# B&R Automation Studio project TD52 (part 86)

#### DirAirInj.var - Local variables
```iecst
(********************************************************************
 * COPYRIGHT -- INNIO Company
 ********************************************************************
 * Program: DirectAirInjection
 * File: DirectAirInjection.var
 * Author: 212754567
 * Created: May 15, 2019
 ********************************************************************
 * Local variables of program DirectAirInjection
 ********************************************************************)

VAR
	xDTGetTime : DTGetTime;
	iDAI_Sec_Act : UDINT; (* direct air injection actual operation time [s] *)
	DT_DAI_Start : DATE_AND_TIME; (* direct air injection starting date and time *)
	xTON_DAI_V_Open_Fault : TON; (* direct air injection inlet valve opening fault delay*)
	xTON_DAI_V_Close_Fault : TON; (* direct air injection inlet valve closing fault delay*)
	xSR_DAI_V_Close_Fault : SR; (* set/reset close fault for direct air injection inlet valve *)
	xSR_DAI_V_Open_Fault : SR; (* set/reset open fault for direct air injection inlet valve *)
	xTOF_DAI_V_Dem : TOF; (* shutdown delay for shut off valve *)
	xTOF_Pr_AirStarter_Tank_Lo : TOF; (* delay enable signal from start tank pressure *)
END_VAR

VAR CONSTANT

END_VAR
```

### Program Logical/EngineController/misf_ctr_EC (IEC) - + misfire monitoring and power reduction

- misf_ctr.st (not readable text: treated as protected, skipped)

#### misf_ctr.var
```iecst
VAR
	bMisfElectrical : BOOL; (* memory for electrical misfire *)
	slMisfIntern : DINT; (* internal integrator for el. misf. *)
	TP_MisfBlink : TP; (* blink pulse for visu. misfiring *)
	ssMisfInt : INT;
	TON_Misfire_Relase : TON;
END_VAR
```

### Program Logical/EngineController/misf_det_EC (IEC) - + detection of misfire using actual power

- misf_det.st (not readable text: treated as protected, skipped)

#### misf_det.var
```iecst
VAR
	ssPowerAuss1 : INT; (* last actual power in permill nom. *)
	FILTER_ActPower : FILTER; (* FUB filter actual power T=30 msec. *)
	bNewAuss : BOOL; (* TRUE= new misfire can be detected *)
	slHilf1 : DINT; (* max.zul.Steilheit von P_ist KW/sec *)
END_VAR
```

### Program Logical/EngineController/MsgEC (IEC) - + Engine Controller Messages

- MsgECCyclic.st (not readable text: treated as protected, skipped)

- MsgECInit.st (not readable text: treated as protected, skipped)

#### MsgEC.var
```iecst
VAR
	iAdrMM2AmmBase : UDINT;
	iAdrAmmBase2MM : UDINT;
	xMsg1080 : Msg;
	xMsg3217 : Msg;
	xMsg1044 : Msg;
	xMsg1049 : Msg;
	xMsg1153 : Msg;
	xMsg3542 : Msg;
	xMsg2061 : Msg;
	xMsg2062 : Msg;
	xMsg2063 : Msg;
	xMsg2064 : Msg;
	xMsg2065 : Msg;
	xMsg2066 : Msg;
	xMsg2067 : Msg;
	xMsg2068 : Msg;
	xMsg2069 : Msg;
	xMsg2070 : Msg;
	xMsg2071 : Msg;
	xMsg2072 : Msg;
	xMsg2073 : Msg;
	xMsg2074 : Msg;
	xMsg2075 : Msg;
	xMsg2076 : Msg;
	xMsg2077 : Msg;
	xMsg2078 : Msg;
	xMsg2079 : Msg;
	xMsg2080 : Msg;
	xMsg2339 : Msg;
	xMsg2365 : Msg;
	xMsg3408 : Msg;
	xMsg3409 : Msg;
	xTON_FG_MSATM : TON;
	FG_MSATM : BOOL;
	xMsg1047 : Msg;
	xMsg3212 : Msg;
	xMsg3099 : Msg;
	xMsg2084 : Msg;
	xMsg1192 : Msg;
	xMsg2514 : Msg;
	xMsg2515 : Msg;
	xMsg2516 : Msg;
	xMsg2517 : Msg;
	xMsg2522 : Msg;
	xMsg2523 : Msg;
	xMsg3348 : Msg;
	xMsg3583 : Msg;
	xMsg3584 : Msg;
	xMsg3529 : Msg;
	xMsg3585 : Msg;
	xMsg3564 : Msg;
	xMsg3371 : Msg;
	xMsg3372 : Msg;
	xMsg3373 : Msg;
	xMsg3374 : Msg;
	bRPSA7_624 : BOOL;
	xTOF_1080_rel : TOF;
	xMsg3586 : Msg;
	FG_ABMW : BOOL; (*Freigabe Abweichung Mittelwert*)
	ton_ABMW : TON;
	xMsg2294 : Msg;
	xMsg2283 : Msg;
	xMsg9216 : Msg;
	xMsg2287 : Msg;
	xMsg2290 : Msg;
	xMsg2262 : Msg;
	xMsg2282 : Msg;
	xMsg2274 : Msg;
	xMsg2588 : Msg;
	xMsg2577 : Msg;
	xMsg2583 : Msg;
	b2880 : BOOL;
	b2881 : BOOL;
	i : USINT;
	iNum_b2880 : USINT;
	iNum_b2881 : USINT;
	xMsg3382 : Msg;
	xMsg2518 : Msg;
	xMsg2519 : Msg;
	xMsg2520 : Msg;
	xMsg2521 : Msg;
	xMsg2562 : Msg;
	xMsg3555 : Msg;
	xMsg3556 : Msg;
	xMsg3557 : Msg;
	xMsg3558 : Msg;
	xMsg2470 : Msg;
	xMsg2471 : Msg;
	xMsg2487 : Msg; (*warning for recommend leanox adjustment*)
	xMsg2488 : Msg; (*warning for mandatory leanox adjustment*)
	xMsg9246 : Msg;
	xMsg2328 : Msg;
	xMsg2329 : Msg;
	xMsg9247 : Msg;
	xMsg9248 : Msg;
	xMsg9253 : Msg; (*warning for Leanox 2 saturation *)
	xMsg9288 : Msg; (* warning: measuring signal failure, temperature direct air injection *)
	xMsg9289 : Msg; (* warning: measuring signal failure, pressure before direct air injection shut off valve  *)
	xMsg9290 : Msg; (* warning: measuring signal failure, pressure before direct air injection control valve bank A *)
	xMsg9291 : Msg; (* warning: measuring signal failure, pressure before direct air injection control valve bank B *)
	xMsg9292 : Msg; (* warning: direct air injection shut off valve failure at closing*)
	xMsg9293 : Msg; (* warning: direct air injection shut off valve failure at opening*)
	xMsg9294 : Msg; (* warning: direct air injection circuit breaker tripped  *)
	xMsg9295 : Msg; (* warning: direct air injection tank pressure low*)
	xMsg9296 : Msg; (* warning: direct air injection control valve bank A failure *)
	xMsg9297 : Msg; (* warning: direct air injection control valve bank B failure *)
	xMsg9298 : Msg; (* warning: direct air injection pressure before shut off valve high *)
	xMsg9299 : Msg; (* warning: direct air injection failure *)
	xMsg9039 : Msg; (* warning: direct air injection active*)
	xMsg9040 : Msg; (* warning: direct air injection inactive*)
	xMsg9312 : Msg; (* Generator frequency too low in mains parallel operation *)
	xMsg9313 : Msg; (* Generator frequency too high in mains parallel operation *)
	xMsg9329 : Msg; (* p2 sensor signal for GEN2 controller missing *)
	xMsg2975 : Msg; (* Fast-Gas-Quality-Change-Function is running *)
	xMsg9047 : Msg; (* operating message: target load reached *)
	xMsg9349 : Msg; (* Grid Code FRT functionality contains wrong parameter *)
	xMsg9053 : Msg; (* operating message: SCR inlet temperature controller active *)
	xMsg9054 : Msg; (* operating message: SCR inlet temperature controller inactive *)
	xMsg9055 : Msg; (* operating message: th. reactor start time reduction - operating cycle started *)
	xMsg9056 : Msg; (* operating message: th. reactor start time reduction - operating cycle completed *)
	xMsg9065 : Msg; (* operating message: Isolated operation - Grid status detection *)
	xMsg9095 : Msg; (* operating message: GEN2 lambda offset stopped *)
	xMsg2765 : Msg; (* warning: PI optimizer opening duration offset in limitation *)
	xMsg3268 : Msg; (* operating message: PI optimizer opening duration offset in limitation *)
	xMsg9373 : Msg; (* warning: PI-Optimization not allowed *)
	xMsg9078 : Msg; (* operating message: PI-Optimization not allowed *)
	xMsg2768 : Msg; (* gas humidity measuring signal failure *)
	xMsg2880 : Msg;	(** B2880: Cylinder exhaust gas temperature positive deviation from average value *)
	xMsg2881 : Msg;	(** B2881: Cylinder exhaust gas temperature negative deviation from average value *)
	xMsg2970 : Msg;	(** B2970: Exhaust gas temperature inclination maximum at cylinder head *)
	xMsg1293 : Msg;	(** B1293: Engine map automatically loaded *)
	xMsg2814 : Msg;	(** B2814: Open durance Port Injection high *)
	xMsg2874 : Msg;	(** B2874: Safety layer sensor failure *)
	xMsg2802 : Msg;	(** B2802: Cylinder pressure sensor measuring signal failure *)
	xMsg2808 : Msg;	(** B2808: Maximum positive deviation of average cylinder peak pressure *)
	xMsg2825 : Msg;	(** B2825: Cylinder peak pressure high Warning *)
	xMsg2826 : Msg;	(** B2826: Cylinder peak pressure high *)
	xMsg2849 : Msg;	(** B2849: Misfiring failure *)
	xMsg2145 : Msg;	(** B2145: Ignition point reduction PBC *)
	xMsg2876 : Msg;	(** B2876: Misfire controller shutdown *)
	xMsg2882 : Msg;	(** B2882: Balancer map deleted *)
	xMsg2883 : Msg;	(** B2883: Balancer map saved *)
	xMsg2960 : Msg;	(** B2960: Ignition point reduction by Cylinder Peak Pressure Integrator *)
	xMsg2141 : Msg;	(** B2141: ignition point optimization *)
	xMsg3238 : Msg;	(** B3238: Positive deviation of cylinder x from average high *)
	xMsg3239 : Msg;	(** B3239: Negative deviation of cylinder x from average high *)
	xMsg3247 : Msg;	(** B3247: TECJET step of gas volume high *)
	xMsg3248 : Msg;	(** B3248: TECJET fuel gas volume high *)
	xMsg3285 : Msg;	(** B3285: exh. gas temp. measuring signal failure *)
	xMsg3295 : Msg;	(** B3295: operation message max. exhaust temperature *)
	xMsg2831 : Msg;	(** B2831: Low Voltage Ride Through Event  --> bBM_GrC_Event *)
	xMsg2832 : Msg;	(** B2832: Mains failure + Generator Pole slip -->  bBM_PoleSlip *)
	xMsg2833 : Msg;	(** B2833: Mains failure + dynamic rotor angle maximum --> bBM_disconnect_dynAng*)
	xMsg2834 : Msg;	(** B2834: Mains failure + static rotor angle maximum -->  bBM_disconnect_staticAng*)
	xMsg2835 : Msg;	(** B2835: Mains failure + leading power factor operation -->bBM_disconnect_CapMode*)
	xMsg2836 : Msg;	(** B2836: Mains failure maintenance request, reserve *)
	xMsg2837 : Msg;	(** B2837: Mains failure + dynamic rotor angle minimum --> bBM_disconnect_dynAng_Min*)
	xMsg2838 : Msg;	(** B2838: Mains failure + electric power to low --> bBM_disconnect_Power*)
	xMsg2839 : Msg;	(** B2839: Mains failure + U(t)< *)
	xMsg9068 : Msg;	(** B9068: Fault ride trougth event  --> bBM_FRT_Event *)
	xMsg9071 : Msg;	(** B9071: Low Voltage Ride Through Event simulated --> bBM_GrC_Event_Sim *)
	xMsg2840 : Msg;	(** B2840: Spare *)
	xMsg2841 : Msg;	(** B2841: Emergency shutdown on gas valves *)
	xMsg2846 : Msg;	(** B2846: Fast power reduction due to auto-ignition *)
	xMsg2852 : Msg;	(** B2852: Turbocharger surge *)
	xMsg2165 : Msg;	(** B2165: Power limitation by air humidity - low limit *)(* Humidity Package *)
	xMsg2166 : Msg;	(** B2166: Air humidity charge temperature offset active *)(* Humidity Package *)
	xMsg2894 : Msg;	(** B2894: Engine map is missing *)
	xMsg1294 : Msg;	(** B1294: performing WG check *)
	xMsg1299 : Msg;	(** B1299: optimizer map changed *)
	xMsg2187 : Msg;	(** B2187: Commissioning mode on *)
	xMsg2188 : Msg;	(** B2188: Commissioning mode off *)
	xMsg2897 : Msg;	(** B2897: Boost pressure out of range*)
	xMsg2929 : Msg;	(** B2929: Cylinder IMEP deviation from average value *)
	xMsg2930 : Msg;	(** B2930: PI optimization required *)
	xMsg2937 : Msg;	(* B2937 LEANOX new adjusted *)
	xMsg2938 : Msg;	(* B2938 Combustion chamber cleaning performed *)
	xMsg2986 : Msg;	(* B2986 Leanox 2 Active - operator message *)
	xMsg2987 : Msg;	(* B2987 Leanox 2 Not Active - operator message *)
	xMsg9388 : Msg; (* warning: combustion anomaly detected *)
	xMsg9392 : Msg; (*warning: CAN wastegate bank A Actuator Failure *)
	xMsg9393 : Msg; (*warning: CAN wastegate bank B Actuator Failure *)
	xMsg9394 : Msg; (*warning: CAN wastegate bank A System Warnings *)
	xMsg9395 : Msg; (*warning: CAN wastegate bank B System Warnings *)
	xMsg2380 : Msg; (*alarm: CAN wastegate bank A CAN Communication Error *)
	xMsg2381 : Msg; (*alarm: CAN wastegate bank B CAN Communication Error *)
END_VAR
```

### Program Logical/EngineController/OUT_EC_TC1 (IEC) - + Engine Controller output task TC1

- OUT_EC_TC1.st (not readable text: treated as protected, skipped)

### Program Logical/EngineController/OUT_EngCtr (IEC) - + Engine Controller output task

- OUT_EngCtr.st (not readable text: treated as protected, skipped)

### Program Logical/EngineController/exhaust_EC (IEC) - + monitoring the exhaust gas temperatures

- exhaustCyclic.st (not readable text: treated as protected, skipped)

- exhaustInit.st (not readable text: treated as protected, skipped)

#### exhaust.var
```iecst
VAR
	FilterCylTemp : ARRAY[0..24] OF FILTER;
	CylTemp_1 : ARRAY[0..24] OF INT;
	ssDeltaCylTemp : INT;
	ABMWN_acttime : ARRAY[0..24] OF UINT; (* 1 hour timer neg. avg. dev. *)
	ABMWN_time : ARRAY[0..24] OF tABMW_time; (* error time memory neg. avg. dev. *)
	ABMWP_acttime : ARRAY[0..24] OF UINT; (* 1 nhour timer pos. avg. dev. *)
	ABMWP_time : ARRAY[0..24] OF tABMW_time; (* error time memory pos. avg. dev. *)
	AmmSeqABMWN : AmmSequence; (* FUB AmmSeq. neg. dev. avg. *)
	AmmSeqABMWP : AmmSequence; (* FUB AmmSeq. pos. dev. avg *)
	AmmSeqATMA : AmmSequence;
	AmmSeqMSAGT : AmmSequence;
	slTempAverage : DINT; (* sum up for average temp. *)
	ssTempLimitNeg : INT; (* cyl.temp. limit negative *)
	ssTempLimitPos : INT; (* cyl.temp. limit positive *)
	ssTempZylMax : INT; (* cyl.temp. maximum value *)
	ssTempZylMin : INT; (* cyl.temp. minimum value *)
	t_zylMax : INT; (* maximal temp. accord. to AN_GW40 *)
	TON_ABMWN : TON; (*reset timer for neg. avg. dev.*)
	TON_ABMWP : TON; (*reset timer for pos. avg. dev.*)
	TON_CheckTemp : TON; (* delay of exh.temp. monitoring *)
	TON_Cycle : TON; (* cycle time for program duration *)
	ucABMWNCount : USINT; (* nbr. of cyl. with neg. deviation *)
	ucABMWPCount : USINT; (* nr. of cyl. with pos. deviation *)
	ucAnzahlZylABWMN : USINT; (* number of cyl. with divagance neg. *)
	ucAverageCount : USINT; (* average # of cylinder counter *)
	ucCylinderCount : USINT; (* cylinder number counter for loops *)
	ucTimeCount : USINT; (* loop counter time memory *)
	usABMWNtime : UINT; (* 1 hour timer neg. avg. dev. *)
	usABMWPtime : UINT; (* 1 hour timer pos. avg. dev. *)
	usTempMaxCount : ARRAY[0..24] OF USINT; (* counter delay max. cyl. temp. *)
	usTempNegCount : ARRAY[0..24] OF USINT; (* counter delay of neg. deviation *)
	usTempPosCount : ARRAY[0..24] OF USINT; (* counter delay of pos. deviation *)
	xHys_EGT_Avg : GR_MAXR;
	xRamp_PRed_EGT_Avg : RAMPE_R;
	t_zyl_mw : INT;
	TOF_HiContSkip : ARRAY[0..25] OF TOF;
	xSimPID_EGT : SimPID4 := (0);
	LCRScal_EG_Max : LCRScal;
	FILTER_EG_Max : FILTER_R;
	TP_ExhLim_FS : TP;
	TON_TempMax_Ext : ARRAY[0..24] OF TON;
	xTON_TempMax_Ext_TrStRed : ARRAY[0..24] OF TON;
	bEngine_Stopped : BOOL;
	TP_bZylAusfall : TP;
	t_zyl_old : ARRAY[0..24] OF INT;
	bEG_Grad : ARRAY[0..24] OF BOOL;
	rT_dTExhMon_ITPComp : REAL; (*TExh compensation at later ITP values (positive values for increasing temp. at retarding) [K/Â°CA]*)
	bdTExhMonTrip : ARRAY[0..24] OF BOOL; (*TRUE = TExhMon trip detected for cylinder*)
	rTsample : REAL; (*task sample time*)
	rdTExh_Misfire : REAL := 20; (*delta temperature from reference to misfire limit [°C]*)
	AmmSeqdTExhMon : AmmSequence;
	bPCGVmonInit : BOOL;
	iCnt_PCGV_class1_Mem : ARRAY[0..24] OF UINT;
	iCnt_PCGV_class2_Mem : ARRAY[0..24] OF UINT;
	iCnt_PCGV_class3_Mem : ARRAY[0..24] OF UINT;
	iCnt_PCGV_class4_Mem : ARRAY[0..24] OF UINT;
	xGR_MINR_t_zyl : ARRAY[0..24] OF GR_MINR;
	xR_TRIG_EGT_PRed : R_TRIG;
	bMSAGT_Warn : ARRAY[0..24] OF BOOL; (*Set the exhaust gas temperature sensor warning*)
	xFILTER_EG_Cyl : ARRAY[0..24] OF FILTER_R;
	iFilt_EG_Cyl : UINT := 5;
	rFILTER_EG_Cyl_old : ARRAY[0..24] OF REAL;
	xGR_MAXR_t_zyl_BackfPrev : ARRAY[0..24] OF GR_MAXR;
	rT_EG_Grad_Hyst : REAL := 0;
	xTP_Ena_BackfPrev : TP;
	rPos_CBV_Release_BackfPrev : REAL := 0.05;
	xMEDIAN_EG_Filt : RMEDIAN24 := (0);
	rGrad_EG_Median : REAL;
	rGrad_EG_Median_old : REAL;
	xTON_t_zyl_BackfPrev : ARRAY[0..24] OF TON;
	tiBackPrevOnDelay : TIME := T#3s;
	rGrad_EG_Filt : ARRAY[0..24] OF REAL;
	rGrad_EG_Filt_Diff2Median : ARRAY[0..24] OF REAL;
	rGrad_EG_Median_Vect : ARRAY[0..24] OF REAL;
	xF_TRIG_bHoldBackfPrev : F_TRIG;
	bBlockBackfPrev : BOOL;
	rP_Act_Norm_BackfPrevOFF : REAL := 0.8;
	bW9388_Array1 : ARRAY[0..24] OF BOOL;
	bW9388_Array2 : ARRAY[0..24] OF BOOL;
	bW9388_Array_Compare : ARRAY[0..24] OF BOOL;
	AmmSeqCombAnomaly : AmmSequence;
	xR_TRIG_bW9388_Array : R_TRIG;
	ucEventCounter : USINT; (*Event counter for loops *)
	xTOF_ZylAusfall : ARRAY[0..20] OF TOF := [21((0))]; (*Timer für Events Zylinderausfall*)
	bTrigZylAusfall : BOOL := 0;
	iZylAusfallErrCout : INT := 0;
	bZylAusfall_test : BOOL := 0;
	rTi_EGT_NegDev : REAL := 180.0; (*Exhaust temperature negative deviation max. duration*)
	rTi_EGT_NegDev_TimeDur : REAL := 180.0; (*Exhauxt temperature negaitve deviation monitoring time duration*)
	iCnt_EGT_NegDev_max : INT := 10; (*Exhaust temperature negative deviation max. count*)
END_VAR
```

### Program Logical/EngineController/dyn_GR (IEC) - + GridCode

- Dyn_GRCyclic.st (not readable text: treated as protected, skipped)

- Dyn_GRInit.st (not readable text: treated as protected, skipped)

#### Dyn_GR.var - Local variables
```iecst
(********************************************************************
 * COPYRIGHT -- INNIO Company
 ********************************************************************
 * Program: dyn_GR
 * File:
 * Author:
 * Created:
 ********************************************************************
 * Local variables of program
 ********************************************************************)
VAR
	bSimulate : BOOL; (*simulation variable*) (* OldName: bSimulate; Cycle:2; *)
	xF_TRIG_IgnOFF : F_TRIG; (* 0 *) (* OldName: F_TRIG_IgnOFF; Cycle:2; *)
	xF_TRIG_VoltRecovPlusT : F_TRIG; (* 0 *) (* OldName: F_TRIG_VoltRecovPlusT; Cycle:2; *)
	xF_TRIG_GCEventPeriode_PA : F_TRIG; (* 0 *) (* OldName: F_TRIG_GCEventPeriode_PA; Cycle:2; *)
	xF_TRIG_GCEvent : F_TRIG; (* 0 *) (* OldName: F_TRIG_GCEvent; Cycle:2; *)
	rN_GrC_Speed : REAL; (* speed for Grid Code calculations *) (* OldName: ssGridCodeSpeed; Cycle:2; *)
	rI_GrC_Lim : REAL; (* Grid Code current limit in [A ]*) (* OldName: ssCurrentLimit; Cycle:2; *)
	rPhase_Ang_Const : REAL; (* constant for phase angel calculation *) (* OldName: fPhaseAngleConst; Cycle:2; *)
	rN_GrC_SpeedChange_Lim : REAL; (* speed change limit for Grid Code event detection *) (* OldName: ssGridCodeSpeedChangeLimit; Cycle:2; *)
	r_Eng_Cyc : REAL; (* Length of motor cycle [ms]*) (* OldName: ssMotorzyklus; Cycle:2; *)
	rU_GrC_Lim : REAL; (* Grid Code voltage limit in [V ]*) (* OldName: ssVoltageLimit; Cycle:2; *)
	rN_Ign_Int : REAL; (* speed ignition [1/min] *) (* OldName: n_Ign_INTERNAL; Cycle:2; *)
	xR_TRIG_IgnOFFON : R_TRIG; (* 0 *) (* OldName: R_TRIG_IgnOFFON; Cycle:2; *)
	xR_TRIG_IgnOFF : R_TRIG; (* 0 *) (* OldName: R_TRIG_IgnOFF; Cycle:2; *)
	xR_TRIG_Wait : R_TRIG; (* 0 *) (* OldName: R_TRIG_Wart; Cycle:2; *)
	xR_TRIG_GCE_Power : R_TRIG; (* 0 *) (* OldName: R_TRIG_GCE_Power; Cycle:2; *)
	xR_TRIG_GCE : R_TRIG; (* 0 *) (* OldName: R_TRIG_GCE; Cycle:2; *)
	xR_TRIG_GCEvent : R_TRIG; (* 0 *) (* OldName: R_TRIG_GCEvent; Cycle:2; *)
	tLam_Ada : TIME; (* 0 *) (* OldName: tLambdaAdabt; Cycle:2; *)
	tLeanoxCtrMan : TIME; (* 0 *) (* OldName: tLeanoxCtrMan; Cycle:2; *)
	tEventPulse : TIME; (* Pulse time for Grid Code event *) (* OldName: tEventPulse; Cycle:2; *)
	tHilfsbetriebeTripOFF : TIME; (* 0 *) (* OldName: tHilfsbetriebeTripOFF; Cycle:2; *)
	tPumpErk : TIME; (* Dauer fuer Aktivierung der Pumperkennung *) (* OldName: tPumpErk; Cycle:2; *)
	tTimeAfterVoltRecov : TIME; (* Zeit nach der, nach Wiederkehr der Spannung, die Zuendung eingeschaltet wird *) (* OldName: tTimeAfterVoltRecov; Cycle:2; *)
	tLeanoxErrorOFF : TIME; (* tLeanoxErrorOFF : TIME; *) (* OldName: tLeanoxErrorOFF; Cycle:2; *)
	tPowerFIX : TIME; (* Dauer Leistungsfixierung bei GCEvent / time Power setting *) (* OldName: tPowerFIX; Cycle:2; *)
	xTOF_GCEventPeriode_PA : TOF; (* *) (* OldName: TOF_GCEventPeriode_PA; Cycle:2; *)
	xTOF_GrC_EventPeriode : TOF; (* No phase angle reset for 1 sec. in case of Grid Code event *) (* OldName: TOF_GirdCodeEventPeriode; Cycle:2; *)
	xTOF_Netp : TOF; (* wait 5 sec. after disconnection from grid to disable the simulation flag *) (* OldName: TOF_Netp; Cycle:2; *)
	xTON_Netp : TON; (* wait 5 sec, after switch to netprallel before use average speed *) (* OldName: xTON_Netp; Cycle:2; *)
	xTON_PoleSlip : TON; (* 0 *) (* OldName: xTON_PoleSlip; Cycle:2; *)
	xTON_ConstGenPF : TON; (* TON check const generator power factor *) (* OldName: TON_ConstGenPF; Cycle:2; *)
	xTON_AvgPeriode : TON; (* time period for average calculation *) (* OldName: TON_AvgPeriode; Cycle:2; *)
	xTON_ConstGenCurr : TON; (*TON check const generator current *) (* OldName: TON_ConstGenCurr; Cycle:2; *)
	xTON_ConstGenFreq : TON; (* 0 *) (* OldName: TON_ConstGenFreq; Cycle:2; *)
	xTP_GrC_Event : TP; (* 0 *) (* OldName: TP_GridCodeEvent; Cycle:2; *)
	xTP_GrC_Event_BM : TP; (* 0 *) (* OldName: TP_GridCodeEvent_BM; Cycle:2; *)
	xTP_GrC_Event_Sim_BM : TP; (* 0 *)
	xTP_GCE_PumpErk : TP; (* 0 *) (* OldName: TP_GCE_PumpErk; Cycle:2; *)
	xTP_GCE_LeanoxErr : TP; (* 0 *) (* OldName: TP_GCE_LeanoxErr; Cycle:2; *)
	xTP_GCE_PowerFIX : TP; (* 0 *) (* OldName: TP_GCE_PowerFIX; Cycle:2; *)
	xTP_VoltRecov : TP; (* 0 *) (* OldName: TP_VoltRecov; Cycle:2; *)
	xTP_Wart : TP; (* 0 *) (* OldName: TP_Wart; Cycle:2; *)
	xTP_PoleSlip : TP; (* 0 *) (* OldName: TP_PoleSlip; Cycle:2; *)
	xTP_IgnOffPump : TP; (* 0 *) (* OldName: TP_IgnOffPump; Cycle:2; *)
	xTP_IgnOnVoltRecov : TP; (* 0 *) (* OldName: TP_IgnOnVoltRecov ; Cycle:2; *)
	xTP_GCE_LeanoxCtr : TP; (* 0 *) (* OldName: TP_GCE_LeanoxCtr; Cycle:2; *)
	xTP_Disc_dynAng_Min_BM : TP; (* 0 *) (* OldName: TP_disconnect_dynAngle_Min_BM; Cycle:2; *)
	xTP_Disc_Power_BM : TP; (* 0 *) (* OldName: TP_disconnect_Power_BM; Cycle:2; *)
	xTP_Disc_dynAng_BM : TP; (* 0 *) (* OldName: TP_disconnect_dynAngle_BM; Cycle:2; *)
	xTP_GCE_Power : TP; (* 0 *) (* OldName: TP_GCE_Power; Cycle:2; *)
	xTP_Disc_CapMode_BM : TP; (* 0 *) (* OldName: TP_disconnect_CapMode_BM; Cycle:2; *)
	xTP_GCE_HBTrip : TP; (* 0 *) (* OldName: TP_GCE_HBTrip; Cycle:2; *)
	xTP_GCE_Lam_Ada : TP; (* 0 *) (* OldName: TP_GCE_LambdaAdabt; Cycle:2; *)
	xTP_GCE : TP; (* 0 *) (* OldName: TP_GCE; Cycle:2; *)
	xTP_DO_GRIDCODE_DCON_TC1 : TP; (* 0 *) (* OldName: TP_DO_GRIDCODE_DCON_TC1; Cycle:2; *)
	xTP_Disc_staticAng_BM : TP; (* 0 *) (* OldName: TP_disconnect_staticAngle_BM; Cycle:2; *)
	xTP_GCE_FIXAct : TP; (* 0 *) (* OldName: TP_GCE_FIXAct; Cycle:2; *)
	xTP_CurrentChange : TP; (* 0 *) (* OldName: TP_CurrentChange; Cycle:2; *)
	xTP_SpeedChange : TP; (* 0 *) (* OldName: TP_SpeedChange; Cycle:2; *)
	xTP_VoltageLow : TP; (* 0 *) (* OldName: TP_VoltageLow; Cycle:2; *)
	b_GrC_VoltageLow : BOOL; (* TRUE if Grid Code event low voltage is detected *) (* OldName: TP_VoltRecov; Cycle:2; *)
	bRel_PA_RESET : BOOL; (* TRUE = PA after 350ms reset *) (* OldName: bFREIGABE_PA_RESET; Cycle:2; *)
	bGrC_Disc_Cap : BOOL; (* Decoupling when capacitance operating in Grid Code Event *) (* OldName: bGC_disconnect_Cap; Cycle:2; *)
	bGrC_Disc_DynAng : BOOL; (* Decouple when static + dynamic angle during GCEvents> Limit*) (* OldName: bGC_disconnect_DynAngle; Cycle:2; *)
	bGrC_Disc_DynAng_Min : BOOL; (* Decouple when static + dynamic angle during GCEvents <Limit*(-1) and voltage below Limi *) (* OldName: bGC_disconnect_DynAngle_Min; Cycle:2; *)
	bGrC_Disc_Power : BOOL; (* Decouple when power < Limit when entering the GC events *) (* OldName: bGC_disconnect_Power; Cycle:2; *)
	bGrC_Disc_StaticAng : BOOL; (* Decouple when static angle already when entering the GC Events> Limit *) (* OldName: bGC_disconnect_StaticAngle; Cycle:2; *)
	bGrC_DO_int : BOOL; (* 0 *) (* OldName: bGC_DO_int; Cycle:2; *)
	bGrC_LamAdabt : BOOL; (* TRUE = Lambda-Adaption aktiv (BR<6) bei BR6 sowieso aktiv LVIC Gasmengenberechnung *) (* OldName: bGC_LambdaAdabt; Cycle:2; *)
	bGrC_LeanoxCtrMAN : BOOL; (* TRUE = Leanox Regler ist im Handbetrieb (GCEvent) *) (* OldName: bGC_LeanoxCtrMAN; Cycle:2; *)
	bGrC_LeanoxCtrMan : BOOL; (* TRUE = Leanox Regler bei GCEvent fuer def. Zeit in Hand *) (* OldName: bGC_LeanoxCtrMan; Cycle:2; *)
	bGrC_LeanoxErrOFF : BOOL; (* TRUE = LoxAbw. A1080 wird bei GCEvent blockiert *) (* OldName: bGC_LeanoxErrOFF; Cycle:2; *)
	bGrC_PowerFIX_Akt : BOOL; (* TRUE = Leistungsfixierung bei GridCodeEvent im eng_ctr aktiv *) (* OldName: bGC_PowerFIX_Akt; Cycle:2; *)
	bGrC_CurrentChange : BOOL; (* TRUE if generator current change is above limit *) (* OldName: bGridCodeCurrentChange; Cycle:2; *)
	bGrC_CurrentChange_Mer : BOOL; (*cuurent chagne merker*) (* OldName: bGridCodeCurrentChange_MERKER; Cycle:2; *)
	bGrC_SpeedChange : BOOL; (* TRUE if Grid Code event speed change is detected *) (* OldName: bGridCodeSpeedChange; Cycle:2; *)
	bGrC_SpeedChange_Mer : BOOL; (*speed change merker*) (* OldName: bGridCodeSpeedChange_MERKER; Cycle:2; *)
	bGrC_Missf : BOOL; (* Switch off the ignition active /TRUE = Zuendungausschalten AKTIV *) (* OldName: bGridMissf; Cycle:2; *)
	bIgnOFF_Mer : BOOL; (* Merker fuer Zuendung AUS *) (* OldName: bIgnOFF_MERKER; Cycle:2; *)
	bIgnON_Mer : BOOL; (* Merker fuer Zuendung EIN *) (* OldName: bIgnON_MERKER; Cycle:2; *)
	bCap : BOOL; (* TRUE = capacitive Engine Run *) (* OldName: bKap; Cycle:2; *)
	bNFilter2 : BOOL; (* TRUE = Avg 2 Perioden | FALSE = 3 Perioden *) (* OldName: bNFilter2; Cycle:2; *)
	bPoleSlip : BOOL; (* TRUE if pole slip detected *) (* OldName: bPoleSlip; Cycle:2; *)
	bPoleSlip_INT : BOOL; (*Pole slip detection*) (* OldName: bPoleSlip_INT; Cycle:2; *)
	bTP_GrC_Event : BOOL; (* TP TRUE Grid Code event *) (* OldName: bTP_GridCodeEvent; Cycle:2; *)
	r_CosPhi : REAL; (* generator cos phi *) (* OldName: fCosPhi; Cycle:2; *)
	r_Phi : REAL; (* generator phi in radian *) (* OldName: fPhi; Cycle:2; *)
	r_Divisor : REAL; (* divisor for polar wheel angle calculation *) (* OldName: fDivisor; Cycle:2; *)
	xFILTER_cosphi : FILTER_R; (*Filter fuer Cos Phi - da Messung im Falle eines Events nicht plausibel*) (* OldName: FILTER_cosphi; Cycle:2; *)
	r_PhaseAng_OFF : REAL; (* dyn. Winkel bei dem die Zuendung AUSgeschalten wird [°] *) (* OldName: fPhaseAngelIgnOFF; Cycle:2; *)
	r_PhaseAng_ON : REAL; (* dyn. Winkel bei dem die Zuendung wieder EINgeschalten wird [°] *) (* OldName: fPhaseAngelIgnON; Cycle:2; *)
	r_PolarWheelAng : REAL; (* calcualted polar wheel angle in degree *) (* OldName: fPolarWheelAngle; Cycle:2; *)
	r_PolarWheelAng_GC : REAL; (* 0 *) (* OldName: fPolarWheelAngle_GC; Cycle:2; *)
	r_Xqo : REAL; (* 0 *) (* OldName: fXqo; Cycle:2; *)
	i_IgnOFF_Time : INT; (* Ignition off aktiv, counter wie lange *) (* OldName: IgnOFF_Time; Cycle:2; *)
	i_IgnOFF_TimeMin : INT; (* 0 *) (* OldName: IgnOFF_TimeMIN; Cycle:2; *)
	iMissfCyl_old_GC : UDINT; (* 0 *) (* OldName: MissfCyl_old_GC; Cycle:2; *)
	rN_Ign1_Avg : REAL; (* avarage speed ignition [1/min] *) (* OldName: n_Ign1_Avg; Cycle:2; *)
	rN_Ign1_old : REAL; (* old speed ignition [1/min] *) (* OldName: n_Ign1_old; Cycle:2; *)
	rN_Ign1_old2 : REAL; (* old speed ignition [1/min] *) (* OldName: n_Ign1_old2; Cycle:2; *)
	rN_GrC_SpeedSumm : REAL; (* speed average sample summ *) (* OldName: slGridCodeSpeedSumm; Cycle:2; *)
	rN_AvgSpeed : REAL; (* 100 sample speed average used for phase angle calcualtion *) (* OldName: ssAvgSpeed; Cycle:2; *)
	rN_AvgSpeed1 : REAL; (* ast sample speed average used for phase angle calcualtion *) (* OldName: ssAvgSpeed1; Cycle:2; *)
	rN_AvgSpeed2 : REAL; (* last sample speed average used for phase angle calcualtion *) (* OldName: ssAvgSpeed2; Cycle:2; *)
	rCnT_GrC_CurrentChange_PULSE : REAL; (* current change puls counter *) (* OldName: ssGCCurrentChange_PULSE_COUNTER; Cycle:2; *)
	rI_GrC_CurrentChange_PULSE_Lim : REAL; (* 0 *) (* OldName: ssGCCurrentChange_PULSE_LIMIT; Cycle:2; *)
	rCnt_GrC_SpeedChange_PULSE : REAL; (* 0 *) (* OldName: ssGCSpeedChange_PULSE_COUNTER; Cycle:2; *)
	rN_GrC_SpeedChange_PULSE_Lim : REAL; (* 0 *) (* OldName: ssGCSpeedChange_PULSE_LIMIT; Cycle:2; *)
	rIgn_Cnt_Off : REAL; (* ignition OFF activate / Zuendung AUS aktiv -> zaehlen wie lange *) (* OldName: ssIgnAUS_Countms; Cycle:2; *)
	rCnt_IGN_Off : REAL; (*Counter for ignition OFF / Counter fuer Zuendung AUS *) (* OldName: ssIGNOFF_COUNTER; Cycle:2; *)
	rCnt_IGN_On : REAL; (*Counter for ignition ON / Counter fuer Zuendung EIN *) (* OldName: ssIGNON_COUNTER; Cycle:2; *)
	r_IL1_Change : REAL; (* change of generator current L1 since last task cycle *) (* OldName: ssIL1Change; Cycle:2; *)
	r_IL2_Change : REAL; (* change of generator current L2 since last task cycle *) (* OldName: ssIL2Change; Cycle:2; *)
	r_IL3_Change : REAL; (* change of generator current L3 since last task cycle *) (* OldName: ssIL3Change; Cycle:2; *)
	r_IL1_Last : REAL; (* Generator current phase 1 from last cycle *) (* OldName: ssLastIL1; Cycle:2; *)
	r_IL2_Last : REAL; (* Generator current phase 2 from last cycle *) (* OldName: ssLastIL2; Cycle:2; *)
	r_IL3_Last : REAL; (* Generator current phase 3 from last cycle *) (* OldName: ssLastIL3; Cycle:2; *)
	r_CosPhi_Last : REAL; (* last power factor *) (* OldName: ssLastCosPhi; Cycle:2; *)
	r_GrC_LastSpeed : REAL; (*speed from last cycle *) (* OldName: ssLastGridCodeSpeed; Cycle:2; *)
	r_Freq_Last : REAL; (*last generator frequency *) (* OldName: usLastFreq; Cycle:2; *)
	iSpeedOption : USINT; (*speed options*) (* OldName: ucSpeedOption; Cycle:2; *)
	bGrC_PumpErk : BOOL; (* TRUE = Pumperkennung bei GC Events aktiv *) (* OldName: bGC_PumpErk; Cycle:2; *)
	iMMUSynchFWVers : ARRAY[0..2] OF UINT; (* Firmware version MMUsynch *) (* OldName: usMMUSynchFWVers; Cycle:2; *)
	iFreqConv : UINT; (* Conversion fuer usFreqNenn[1] *) (* OldName: usFreqConv; Cycle:2; *)
	iCnt_Avr : USINT; (* counter for calcualte average of engine speed *) (* OldName: usCounter; Cycle:2; *)
	iSWCycltime : USINT; (* Softwarezykluszeit des GridCode Tasks [ms] *) (* OldName: ucSWCycltime; Cycle:2; *)
	iCnt_GrC_Event_Lim : DINT; (* Limit for mains failure maintenance request *) (* OldName: ucGCEvent_CounterLIMIT; Cycle:2; *)
	iCylOFF_cycl : USINT; (* Max. Anzahl an Motorzyklen fuer Zuendung AUS [Motorzyklen * 10] *) (* OldName: ucCylOFF_cycl; Cycle:2; *)
	iCylON_cycl : USINT; (* Min. Anzahl an Motorzyklen fuer anschliessend Zuendung EIN [Motorzyklen * 10] *) (* OldName: ucCylON_cycl; Cycle:2; *)
	rSpeedChange : REAL; (* speed change since last task cycle *) (* OldName: ssSpeedChange; Cycle:2; *)
	iSpeedMinus : INT; (* Ausloesung Zuendung EIN bei Drehzahl x U/min unter Durchschnittsdrehzahl *) (* OldName: ssSpeedMinus; Cycle:2; *)
	iSpeedMinus2 : INT; (* 0 *) (* OldName: ssSpeedMinus2; Cycle:2; *)
	iSpeedPlus : INT; (* Ausloesung Zuendung AUS bei Drehzahl x U/min ueber Durchschnittsdrehzahl *) (* OldName: ssSpeedPlus; Cycle:2; *)
	iSpeedPlus2 : INT; (* 0 *) (* OldName: ssSpeedPlus2; Cycle:2; *)
	tFIXActuators : TIME; (* 0 *) (* OldName: tFIXActuators; Cycle:2; *)
	bLeanox_Man_old : BOOL; (* leanox controller in manual old *) (* OldName: l_einst_a_old; Cycle:2; *)
	bVoltRecovAct : BOOL; (* TRUE = Zuendung spaetestens ein sobald Spannung wieder da + Zeit | FALSE = Zuendung spaetestens nach "tPulseEvent" ein*) (* OldName: bVoltRecovAct; Cycle:2; *)
	bGC_HilfsbetriebeTripOFF : BOOL; (*TRUE = Stoerung HB (A1129) wird bei GCEvent blockiert*) (*  *)
	iNrOfPolePair : INT; (*amount of pole pairs*)
	bGearBox : BOOL; (*TRUE = GearBox (Motor with 1500U/min in 60Hz Netz)*) (* OldName: ; Cycle: 2 *)
	rF_Calc : REAL;
	FILTER_R_P2s_WP : FILTER_R; (*Filter fuer den p2s Arbeitspunkt bei Eventeintritt*)
	rPr_P2s_t0 : REAL; (*Laderuck gefiltert vor GC-Event (t0)*)
	rPos_CBV_t0 : REAL; (*CBV Position vor GC-EVent (t0)*)
	iT_GrC_1_2 : INT; (*Verzoegerungszeit fuer Oeffnen des CBV [10ms]*)
	iT_GrC : INT; (*Timer [10ms] waehrend dem Event*)
	rDPos_Phase2 : REAL; (*delta CBV Position fuer Phase 2 (oeffnen) )[-]*)
	rDPos_Phase3 : REAL; (*delta CBV Position fuer Phase 3 (schliessen) )[-]*)
	usFilt_P2s_t0 : USINT; (*Filterzeitkonstante fuer die Ermittlung der P2s zum Zeitpunkt t0 [10ms]*)
	usFilt_P2s_tn : USINT; (*Filterzeitkonstante fuer die Ermittlung der P2s waehrend dem Event [10ms] 0 = keine Filterung*)
	FILTER_R_P2s_tn : FILTER_R;
	rPr_P2s_tn : REAL;
	iGrC_Phase_old : INT;
	rPos_TV_t0 : REAL; (*TV Position vor GC-EVent (t0)*)
	rLam_Leanox_Set_t0 : REAL; (*Lambda Wert vor GC-EVent (t0)*)
	rLam_Leanox_Set_GrC : REAL;
	rLamOfs_GrC : REAL;
	bGrC_SimulateEvent : BOOL; (*DO NOT CHANGE!!!*)
	b_RelLamAdapt : BOOL;
	rK_Lam : REAL;
	rmaxdLam : REAL;
	tSimuVLow : TIME := T#250ms;
	TP_SimulateVoltageLow : TP;
	bGrC_SimulateVLow : BOOL;
	b_SIMULATE : BOOL;
	rObereGrenze_p2s : REAL;
	rUntereGrenze_p2s : REAL; (*Untere p2s Grenze fuer An*)
	iGrC_Phase : INT; (*Phase des LVRT Events*)
	bFG_GC_III : BOOL; (*TRUE = GridCode Phase III Funktionen AKTIV*)
	iIgnOffTestMode_t : ARRAY[0..3] OF INT; (*Zeit fuer IgnOffTestMode [10ms] Phase[i]*)
	iIgnOffTestModeCount : INT;
	rdPos_CBV_GrC : REAL; (*Offset fuer Rampe Anfang Phase 2*)
	rRampe_CBV : REAL; (*Rampe fuer CBV in Phase 2[-/100ms]*)
	rPos_CBV_max_GrC : REAL; (*Max. Absolutposition CBV*)
	iUBV_fix : INT; (*Nummer vom zu fixierenden UBV*)
	rPos_CBVfixed : REAL;
	bVorStIgnOFF : BOOL; (*Vorsteuerung IgnOFF bei GC-Event*)
	iVorstIgnOFF : INT; (*Dauer Vorsteuerung IgnOFF bei GC-Event [*10ms]*)
	bVorStIgnON : BOOL; (*Vorsteuerung IgnON bei GC-Event*)
	iVorstIgnON : INT; (*Dauer Vorsteuerung IgnON bei GC-Event [*10ms]*)
	iCountVorstIgnON : INT;
	iCountVorstIgnOFF : INT;
	rcosphiLim_VorstIgn : REAL; (*Cos phi Limit fuer Freigebe der Vorsteuerung Zuendung AUS*)
	rPLim_VorstIgn : REAL; (*Wirkleistungs Limit fuer Freigebe der Vorsteuerung Zuendung AUS bezogen auf die Nennleistung*)
	bVorstIgnAct : BOOL; (*TRUE = Cos phi und Leistungs-Limits fuer Freigabe der Vorsteuerung Zuendung AUS erfuellt*)
	TON_Vorst : TON;
	iGrC_Phase_Old : INT;
	rRampe_CBV_neg : REAL;
	rDPos_Rampe : REAL;
	rU_GrC_Min : REAL; (*min. Spannung Phase - Phase*)
	bVorstIgnAct_U : BOOL;
	rPos_WG_GrCfixed : REAL;
	rPos_WG_t0 : REAL; (*WG Position vor GC-EVent (t0)*)
	bGrC_WG_open_close : BOOL; (*WG bei Event oeffnen - anschliessend komplett schliessen (Prio. 2)*)
	bGrC_WG_open_back : BOOL; (*WG bei Event oeffnen - anschliessend zurueck auf Ausgangswert (Prio. 3)*)
	bGrC_WG_close : BOOL; (*WG bei Event schliessen (Prio. 1)*)
	ucCylinderCount : USINT; (* loop counter number of cylinder *)
	bSIM_HVRT : BOOL;
	bGrC_SimulateVHigh : BOOL;
	rU_GrC_Lim_HVRT : REAL;
	rGrC_Voltage_Lim_HVRT : REAL;
	rN_GrC_SpeedChange_Lim_HVRT : REAL;
	rGrC_SpeedChange_Lim_HVRT : REAL;
	rI_GrC_Lim_HVRT : REAL;
	rGrC_CurChange_Lim_HVRT : REAL;
	b_GrC_VoltageHigh : BOOL;
	bGrC_NChangeHVRT : BOOL;
	bGrC_CurChange_HVRT : BOOL;
	rCnt_GrC_NChange_PULSE_HVRT : REAL;
	rN_GrC_NChange_PULSE_Lim_HVRT : REAL;
	bGrC_NChange_Mer_HVRT : BOOL;
	rCnT_GrC_Cur_PULSE_HVRT : REAL;
	rI_GrC_CurChange_PULSE_Lim_HVRT : REAL;
	bGrC_CurChange_Mer_HVRT : BOOL;
	bGrC_Event_HVRT : BOOL;
	bVorStIgn_simu : BOOL := 0;
	iVorstIgnOFF_simu : INT := 0;
	bGrC_Freeze_HVRT : BOOL := 0;
	bFreeze_at_HVRT : BOOL;
	xTP_GCE_PowerFIX_HVRT : TP;
	bManCBV_Vorgabe : BOOL := 0;
	rDPos_Phase2man : REAL;
	iVorstIgnLATE : INT; (*Dauer Vorsteuerung IgnLATE bei GC-Event [*10ms]*)
	bIGTLatePhase2ON_simu : BOOL := 0;
	bIGTLatePhase2_komplett : BOOL := 0;
	bVorstIgnLATE : BOOL := 0;
	bNO_LEANOX_MAN_GEN2 : BOOL := 0;
	xFILTER_pel : FILTER_R := (0);
	rP_IST_NOM : REAL;
	PF_Act_lin : REAL;
	PF_Act_lin_back : REAL;
	uiFiltercosphi : UINT := 100;
	MisfireCyl : ARRAY[0..24] OF UDINT;
	bReleaseTest : BOOL := 0; (*Aktivierung der Zylinder.Zuendung-Abschaltfunktion*)
	iCylNummer : INT; (*Zylindernummer des 1. Zylinders der abgeschalten werden soll*)
	iCylNummer2 : INT; (*Zylindernummer des 2. Zylinders der abgeschalten werden soll*)
	iZeitLimit : INT := 0; (*Zeit fuer das Abschalten der Zylinder [ms]*)
	iZeitCount : INT;
	iGrC_Phase_CBV : INT; (*Phase of LVRT event for CBV*)
	ti_TON_GrCPhase4 : TIME := T#1s; (* Minimum time before release of CBV in phase 4 *)
	xTON_GrC_Phase4 : TON; (*  TON Minimum time before release of CBV in phase 4 *)
	rOffsetSollWert : REAL; (* PI-Duration setpoint of offset *)
	xSigScalR_rGasFlowDec_GrC : xSigScal_R; (* Interpolation of gas flow factor depending on engine power *)
	rGasFlowDec_GrC : REAL; (* Interpolated gas flow factor depending on engine power *)
	xTOF_ITP_DynGrC : TOF; (* TOF ITP change for dynamic grid code *)
	ti_TOF_ITP_DynGrC : TIME; (* Duration of ITP change for dynamic grid code *)
	rCA_Ign_Act_old : ARRAY[0..24] OF REAL; (* Actual cylinder ignition point before grid event  *)
	xLCRRamp_GrC_Offset : LCRRamp; (* Ramp for gas flow factor *)
	xTOF_rGasflow_Factor_GrC : TOF; (* Holding time of gas flow factor *)
	bTestBit_GasFlowRed_GrC : BOOL; (* Activate gas flow factor for testing *)
	bTestBit_ITP_GrC : BOOL; (* Activate ITP change for testing *)
	rFactor_Gearbox : REAL; (* Factor for gear transmission ratio *)
	xTON_Insel : TON; (* TON for transition to island operation *)
	rN_FRT_SpeedChange_Lim_EPS : REAL; (* Speed change limit for fault ride trough detection in island operation [1/min/s] *)
	rI_FRT_Lim_EPS : REAL; (* Fault ride trough detection current limit in island operation [%Inenn/s] *)
	rU_FRT_Lim_EPS : REAL; (* Fault ride trough detection voltage limit in island operation [%Unenn] *)
	bFRT_VoltageLow_EPS : BOOL; (* TRUE if fault ride trough event low voltage in island operation is detected *)
	rSpeedChange_EPS : REAL; (* Speed change since last task cycle in island operation [rpm] *)
	rN_FRT_LastSpeed_EPS : REAL; (* Speed from last cycle in island operation [rpm] *)
	bFRT_SpeedChange_EPS : BOOL; (* TRUE if fault ride trough speed change in island operation is detected *)
	iCnt_FRT_SpeedChangePULSE_EPS : INT; (* Counter of speed change flag in island operation *)
	iN_FRT_SpeedChangePULSELim_EPS : INT; (* Limit for counter of speed change flag in island operation *)
	bFRT_SpeedChange_Mer_EPS : BOOL; (* Speed change flag in island operation *)
	rIL1_Change_EPS : REAL; (* Change of generator current L1 since last task cycle in island operation [A] *)
	rIL1_Last_EPS : REAL; (* Generator current phase 1 from last cycle in island operation [A] *)
	rIL2_Change_EPS : REAL; (* Change of generator current L2 since last task cycle in island operation [A] *)
	rIL2_Last_EPS : REAL; (* Generator current phase 2 from last cycle in island operation [A] *)
	rIL3_Change_EPS : REAL; (* Change of generator current L3 since last task cycle in island operation [A] *)
	rIL3_Last_EPS : REAL; (* Generator current phase 3 from last cycle in island operation [A] *)
	bFRT_I_Change_EPS : BOOL; (* TRUE if generator current change in island operation is above limit *)
	iCnT_FRT_I_ChangePULSE_EPS : INT; (* Counter of current change flag in island operation *)
	iFRT_I_ChangePULSELim_EPS : INT; (* Limit for counter of current change flag in island operation *)
	bFRT_I_Change_Mer_EPS : BOOL; (* Current change flag in island operation *)
	xTP_FRT_Event_BM : TP; (* TP Fault ride trough in island operation *)
	bPoleSlip_EPS_INT : BOOL; (*Pole slip detection in island operation*)
	bPoleSlip_EPS : BOOL; (* TRUE if pole slip in island operation is detected *)
	xTON_PoleSlip_EPS : TON; (* TON for pole slip detection in island operation *)
	xTP_PoleSlip_EPS : TP; (* TP for pole slip detection in island operation *)
	xTP_FRT_Event_BM_EPS : TP; (* TP for FRT event in island operation *)
	bTestbutton_Deact : BOOL; (* Deactivate the gridcode test buttons for debug *)
	TOF_GrC_Test_150 : TOF; (* TOF start 150ms gridcode test *)
	TOF_GrC_Test_250 : TOF; (* TOF start 250ms gridcode test *)
	TOF_GrC_Test_Var : TOF; (* TOF start variable gridcode test *)
	R_TRIG_GrC_Test : R_TRIG; (* Trigger of dynamic grid code test buttons *)
	iNrOfPoleSlipSinceStart : INT := 0; (* Number of pole slip events since last start *)
	iEngineCycleTime : INT; (* Engine cylce time depending on nominal speed *)
	xTP_DO_GRIDCODE_EPS_DCON_TC1 : TP; (* TP for opening GCB with pole slip detection in island operation *)
	iMissfCyl_FRT_Set : UDINT; (* Set point of switched off cylinders during FRT event *)
	xTOF_FRT_Offset_PI : TOF; (* Delay of PI valve offset after FRT event *)
	bITP_Shift_FRT : BOOL; (* ITP shift during Ignition OFF at FRT event *)
	xRAMPE_R_ITP_FRT : LCRRamp; (* Ramp of ITP set point after FRT event *)
	xTOF_ITP_Ramp_FRT : TOF; (* TOF of active ITP set point ramp *)
	ti_TOF_ITP_Ramp_FRT : TIME; (* Duration of active ITP set point ramp after FRT event *)
	rCA_Ign_Act_Max : REAL; (* Maximum IPT set point of all cylinders when no FRT event is active *)
END_VAR
```

### Program Logical/EngineController/GR_GCB_cust (IEC) - + GridCode Custom

- GR_GCB_custCyclic.st (not readable text: treated as protected, skipped)

#### GR_GCB_cust.var - Local variables
```iecst
(********************************************************************
 * COPYRIGHT -- INNIO Company
 ********************************************************************
 * Program: GR_GRB_cust
 * File: GR_GRB_cust.var
 * Author: 502221015
 * Created: June 27, 2013
 ********************************************************************
 * Local variables of program GR_GRB_cust
 ********************************************************************)
VAR
	xTON_ULo : ARRAY[0..2] OF TON; (* Low Voltage time delay*) (* OldName: TON_10ms_VoltageLow22; Cycle:5; *)
	rU_LxLy_Min : REAL; (* Lowest voltage of all three phases*) (* OldName: bGridCodeVoltageLow22; Cycle:5; *)
	i : INT; (* For-loop counter*) (* OldName: bGridCodeVoltageLow23_200; Cycle:5; *)
	bGrC_ULo_Trig : BOOL; (* Gridcode low voltage trigger*) (* OldName: bGridCodeVoltageLow21_200; Cycle:5; *)
	xTP_ULo : TP; (*   *) (* OldName: TP_10ms_VoltageLOW; Cycle:5; *)
	xTP_ULo_BM : TP; (*   *) (* OldName: TP_10ms_VoltageLOW_BM; Cycle:5; *)
	xTON_F_OverMp : TON; (* TON - Generator protection high frequency W9313 *)
	xTON_F_UnderMp : TON; (* TON - Generator protection low frequency W9312 *)
	rN_Offset_Test : REAL := 0; (* Speed offset for testing purposes *)
	iNrOfPolePair : INT; (* Amount of pole pairs *)
	xTP_DO_GENERATOR_DCON_TC1 : TP; (* GCB opening command of three seconds *)
	rF_GR_Filt_min : REAL := 47; (*minimal filtered grid frequency for leanox/itp adaptation*)
	rF_GR_Filt_max : REAL := 63; (*maximal filtered grid frequency for leanox/itp adaptation*)
	iFactTFilt_N_GR : UINT := 2; (*Grid frequency filter multiplication factor for island mode*)
	bGearBox : BOOL; (* TRUE = GearBox (Engine with 1500rpm @ 60Hz Grid) *)
	rF_Calc : REAL; (* Calculated frequency depending on nominal engine speed *)
	rN_GR_Speed : REAL; (* Speed for Grid Code calculations *)
	xLCRPT1_N_GR : LCRPT1; (*speed filter for static grid code calculations*)
	bGrC_GCB_DCON_ULo : BOOL; (* Open GCB in case of voltage break-in *)
	bGrC_GCB_DCON_Freq : BOOL; (* Open GCB in case low/high frequency *)
END_VAR
```

### Program Logical/EngineController/VisEC (IEC) - + Visualization task

- VisEC.st (not readable text: treated as protected, skipped)

#### VisEC.var - Local variables
```iecst
(********************************************************************
 * COPYRIGHT -- INNIO Company
 ********************************************************************
 * Program: VisEC
 * File: VisEC.var
 * Author: 502423184
 * Created: October 27, 2015
 ********************************************************************
 * Local variables of program VisEC
 ********************************************************************)
VAR
	rT_EG_System : REAL;
	xTON_Load_Delay : TON := (0);
	bOld_RKS_Ena : BOOL;
	bAut_Opt_Act_old : BOOL;
END_VAR
```

### Program Logical/EngineController/ParEC (IEC, version 4.06.0) - + Engine Controller Parameter

- perm_par.st (not readable text: treated as protected, skipped)

#### perm_par.var
```iecst
VAR
	tParaIntern : ParaHandler_typ; (*Connector type to perm_par*)
	tMM2ParaBase_ReadBack : MM2ParaBase_type; (*INTERNAL! V4.06 new readback structure for information from previous tasks*)
	bWriteDataObj : BOOL; (* TRUE=write data object module *)
	bDataObjLenErr : BOOL; (*Error occured in permem: data module size missmatch*)
	bCreateDataObj : BOOL; (* TRUE=create new data object *)
	bWriteOnce : BOOL; (* write permanent memory once *)
	DatObjCreate_01 : DatObjCreate; (* data object create *)
	DatObjInfoBak_02 : DatObjInfo; (* data object info *)
	DatObjDelete_01 : DatObjDelete; (* data object delete *)
	DatObjRead_01 : DatObjRead; (* data object read *)
	DatObjRead_02 : DatObjRead; (* manual initiated data object read *)
	DatObjWrite_01 : DatObjWrite; (* data object write *)
	DatObjDelete_02 : DatObjDelete; (* data object delete *)
	DatObjDelete_11 : DatObjDelete; (*Delete Backup File*)
	DatObjInfo_01 : DatObjInfo; (* data object info *)
	DatObjInfo_02 : DatObjInfo; (* data object info *)
	szModuleName : STRING[35]; (* module name of object *)
	szModuleNameBackup : STRING[35]; (* module name of posiibly created backup object *)
	DatObjCopy_01 : DatObjCopy;
	bCopyDataObj : BOOL;
	TON_WarnDelay : TON;
	TON_WritePMEM : TON; (* delay write permanent memory *)
	ulPMPointer : UDINT; (* adress of actual checksum value *)
	ulChecksum : UDINT; (* parameter checksum value *)
	pm_len : UDINT; (* permanent value lenght *)
	ulChecksumOld : UDINT; (* last vlaue of parameter checksum *)
	ulChkValue : UDINT; (* actual value of parameter pointer *)
	pm_id : UDINT; (* permanent value identifier *)
	pm_p : UDINT; (* permanent value pointer *)
	DatObjInfo_META : DatObjInfo;
	DatObjRead_META : DatObjRead;
	szMetaDataRaw : STRING[2000];
	szMetaData : ARRAY[0..4] OF STRING[35];
	szMetaDataVis : ARRAY[0..3] OF STRING[35];
	ssIndex : INT;
	ssCount : INT;
	ucMetaDataRaw : ARRAY[0..2000] OF USINT;
	ssCount2 : INT;
	szMetaDataFile : STRING[10];
	szText1 : STRING[20];
	pv_adr_IN_XX_tPB2MM : UDINT;
	pv_lng : UDINT;
	pv_lng_IN_XX_tPB2MM : UDINT;
	pv_lng_OUT_XX_tPB2MM : UDINT;
	szText2 : STRING[20];
	pv_adr_OUT_XX_tXX2PB : UDINT;
END_VAR
VAR CONSTANT
	ERR_NOERROR : UINT := 0;
END_VAR
VAR
	usPMWriteCnt : UINT;
	pm_Error : UDINT; (* permanent value error *) (* Deleted: pm : ParaMem_typ; permanent memory tags mathias, 22.8.11*)
	fun_Error : UDINT := 0; (*state > 0 = function error*)
	xLocalParaCheck : ParaCheckFUB; (*local function instance to check parameter values*)
	TON_ParaSetupOk : TON;
	bParaCheckSystemOk : BOOL;
	iDebug_ParaOkChecked : UDINT;
	bRestoreBackupDataObj : BOOL := FALSE;
	bRestoreDataObjContent : BOOL := FALSE;
	pm_id_backup : UDINT;
	pm_p_Backup : UDINT;
	DatObjCopy_02 : DatObjCopy;
	bDeleteBackupDataObj : BOOL := FALSE; (*Command to delete backup data module file on purpose*)
	bDebugPara : ARRAY[0..5] OF BOOL;
	ssIndex2 : INT;
	ssIndex3 : INT;
	ssIndex4 : INT;
	ssIndexVis : INT;
	szText : STRING[40];
	pv_adr_Para : UDINT;
	szParaSnippet : ARRAY[0..5] OF STRING[150];
	szParaIndex : STRING[10];
	slValue : DINT;
	iModuleDLD_ResetCount : INT;
	bDownloadDetected : BOOL;
	bFlagParaStructCopyWorking : BOOL; (*true, if cyclic para copying is active, 1 false cycle at every copy *)
	bStoreInitParaInDataObj : BOOL := FALSE;
	bTestflag : BOOL;
	bReadOutMETA_Once : BOOL;
	tParaCheck_iPvAdress : ARRAY[0..5] OF UDINT;
	tParaCheck_iPvLengt : ARRAY[0..5] OF UDINT;
	tParaCheck_rPvValue : ARRAY[0..5] OF REAL;
	tParaCheck_rRangeMIN : ARRAY[0..5] OF REAL;
	tParaCheck_rRangeMAX : ARRAY[0..5] OF REAL;
	tParaCheck_szPvName : ARRAY[0..5] OF STRING[35];
	ssFormatDetected : INT;
	szMetaDataPart : STRING[150];
	szFullTaskName : STRING[35];
	szFullMetaModuleName : STRING[35];
	debugLen : INT;
	debugSize : INT := 0;
	strcat_adr1 : UDINT;
	strcat_adr2 : UDINT;
	ssIndexTN : INT;
	bAlternate : BOOL;
	n : INT;
	iAlternateChecksum : DINT;
	iAlternateChecksumOld : DINT;
	ulDebugChkValue : ARRAY[0..999] OF UDINT;
	Adr1 : UDINT;
	Adr2 : UDINT;
	usPMWriteCntStepsize : UINT := 1; (*different step sizes to help debug*)
	usPMWriteCntXOR : UINT;
	usPMWriteCntAltSum : UINT;
	ulAdrPM : UDINT;
	usChkValuePM : USINT;
	ulAdrPara : UDINT;
	ulPara_len : UDINT;
	usChkValuePara : USINT;
	iDebugCountPMDifferences : DINT := 0;
	bEngineRunDetected : BOOL; (*detection status bit autocommand 100 /101  for engine run state*)
	ucMetaDataDebugInfoLine : ARRAY[0..24] OF STRING[80];
	ssIndexMand : INT := 0;
	szMetaDataMand : STRING[35];
	iMyErrorInfo_Autoreset : DINT; (*internal autoreset counter*)
	ssIndex_Version : INT; (*internal*)
	ssIndex_BU : INT; (*internal*)
	ssIndex_BU2 : INT; (*internal*)
END_VAR
```

### Program Logical/EngineController/PermMap (IEC) - + Additional Engine Maps

- PermMapCyclic.st (not readable text: treated as protected, skipped)

- PermMapInit.st (not readable text: treated as protected, skipped)

#### PermMap.typ - Local data types
```iecst
(********************************************************************
 * COPYRIGHT -- INNIO Company
 ********************************************************************
 * Program: PermEC
 * File: PermEC.typ
 * Author: WaldharM
 * Created: October 16, 2012
 ********************************************************************
 * Local data types of program PermEC
 ********************************************************************)

TYPE
	ParaMap_typ : 	STRUCT
		Map : Map_Struct;
		Cnt : Cnt_Struct;
	END_STRUCT;
END_TYPE
```

#### PermMap.var - Local variables
```iecst
(********************************************************************
 * COPYRIGHT -- INNIO Company
 ********************************************************************
 * Program: PermEC
 * File: PermEC.var
 * Author: WaldharM
 * Created: October 16, 2012
 ********************************************************************
 * Local variables of program PermEC
 ********************************************************************)
VAR
	pm_Error : UINT;
	write_once : BOOL;
	pm_len : UDINT;
	ModulName : STRING[35];
	DatObjInfo_01 : DatObjInfo;
	pm_id : UDINT;
	pm_p : UDINT;
	bCreateDataObj : BOOL;
	perm_par_vers : UINT;
	DatObjRead_01 : DatObjRead;
	usPMWriteCnt : UINT;
	DatObjDelete_PermMem : DatObjDelete;
	DatObjCreate_01 : DatObjCreate;
	DatObjWrite_01 : DatObjWrite;
	ulChecksumOld : UDINT;
	ulPMPointer : UDINT;
	ulChkValue : UDINT;
	TON_WritePMEM : TON;
	ulChecksum : UDINT;
	bWriteDataObj : BOOL;
END_VAR
VAR CONSTANT
	ERR_NOERROR : UINT := 0;
END_VAR
VAR
	pmm : ParaMap_typ;
	TON_BlockMinFileAge : TON;
	bBlock_MinFileAge : BOOL;
	TP_DemPermSave : TP;
END_VAR
```

### Program Logical/EngineController/PermEC2 (IEC) - + Additional Engine Maps

- PermECCyclic.st (not readable text: treated as protected, skipped)

- PermECInit.st (not readable text: treated as protected, skipped)

#### PermEC.typ - Local data types
```iecst
(********************************************************************
 * COPYRIGHT -- INNIO Company
 ********************************************************************
 * Program: PermEC
 * File: PermEC.typ
 * Author: WaldharM
 * Created: October 16, 2012
 ********************************************************************
 * Local data types of program PermEC
 ********************************************************************)

TYPE
	ParaEC2_typ : 	STRUCT
		Map : Map_Struct;
		Perm : Perm_Struct;
		iCnt_TC_Surge : DINT;
		iCnt_GrCEvent : DINT;
	END_STRUCT;
END_TYPE
```

#### PermEC.var - Local variables
```iecst
(********************************************************************
 * COPYRIGHT -- INNIO Company
 ********************************************************************
 * Program: PermEC
 * File: PermEC.var
 * Author: WaldharM
 * Created: October 16, 2012
 ********************************************************************
 * Local variables of program PermEC
 ********************************************************************)
VAR
	pm_Error : UINT;
	write_once : BOOL;
	pm_len : UDINT;
	ModulName : STRING[35];
	DatObjInfo_01 : DatObjInfo;
	pm_id : UDINT;
	pm_p : UDINT;
	bCreateDataObj : BOOL;
	perm_par_vers : UINT;
	DatObjRead_01 : DatObjRead;
	usPMWriteCnt : UINT;
	DatObjDelete_PermMem : DatObjDelete;
	DatObjCreate_01 : DatObjCreate;
	DatObjWrite_01 : DatObjWrite;
	ulChecksumOld : UDINT;
	ulPMPointer : UDINT;
	ulChkValue : UDINT;
	TON_WritePMEM : TON;
	ulChecksum : UDINT;
	bWriteDataObj : BOOL;
END_VAR
VAR CONSTANT
	ERR_NOERROR : UINT := 0;
END_VAR
VAR
	pmm : ParaEC2_typ;
	TON_BlockMinFileAge : TON;
	bBlock_MinFileAge : BOOL;
END_VAR
```

### Program Logical/EngineController/PVcheckNEW (IEC) - + checks and loads PV's for pre-mixed engines

- PVcheck.st (not readable text: treated as protected, skipped)

#### PVcheck.var - Local variables
```iecst
(********************************************************************
 * COPYRIGHT -- INNIO Company
 ********************************************************************
 * Program: PermINIT
 * File: PermINIT.var
 * Author: 502293141
 * Created: February 24, 2015
 ********************************************************************
 * Local variables of program PermINIT
 ********************************************************************)
VAR
	bSKIP_DataLoad : BOOL;
	bLAMBDA_DataLoad : BOOL;
	bGEN2_DataLoad : BOOL;
	bPSICAL_DataLoad : BOOL;
	bENGCTR_DataLoad : BOOL;
	TON_FGDRPS_MAP : TON;
	bSafety_DataLoad : BOOL;
	bMFB50_Dataload : BOOL;
	bOpt_DataLoad : BOOL;
	bAmmSeqClkP : BOOL;
	TON_SecondTick : TON;
	bMapLoaded : ARRAY[0..24] OF BOOL;
	i : INT;
	bMapLoad : BOOL;
	xTON_Reset : TON := (0);
	bPUSL_DataLoad : BOOL := 0;
	bFilt_DataLoad : BOOL := 0;
	bWG_DataLoad : BOOL;
	bEG_DataLoad : BOOL;
	bAutoLoad_Ena : BOOL;
	TON_AutoLoad : TON;
	bPermFailedNew : ARRAY[0..24] OF BOOL;
	bFS_DataLoad : BOOL;
	bALL_Dataload : BOOL := 0;
	bIG_DataLoad : BOOL := 0;
	bAutoLoad_Ena_TP : BOOL := 0;
	TP_bAutoLoad : TP := (0);
	bSync_DataLoad : BOOL := 0;
	TON_ParaSetupOk_10s : TON;
	iNimmCBV_old : INT;
	bLX2_DataLoad : BOOL;
	bTrStRed_DataLoad : BOOL;
	bVE_CYS	:	BOOL;
	rLCRCurve_DK_min_Lup_y5 : REAL := 0.65; (*containment GEN2 TVmin GridP*)
	rLCRCurve_DK_min_Lup_y6 : REAL := 0.8; (*containment GEN2 TVmin GridP*)
	bGen2_LQR_DataLoad : BOOL;
	bParaLoaded_Gen2_LQR_T9 : BOOL; (* Parameter were loaded for Gen2 LQR T9 *)
END_VAR
```

### Program Logical/EngineController/PVcheck (IEC) - + checks and loads PV's for type 9

- PVcheck.st (not readable text: treated as protected, skipped)

#### PVcheck.var - Local variables
```iecst
(********************************************************************
 * COPYRIGHT -- INNIO Company
 ********************************************************************
 * Program: PermINIT
 * File: PermINIT.var
 * Author: 502293141
 * Created: February 24, 2015
 ********************************************************************
 * Local variables of program PermINIT
 ********************************************************************)
VAR
	bSKIP_DataLoad : BOOL;
	bPI_DataLoad : BOOL;
	bLAMBDA_DataLoad : BOOL;
	bPSICAL_DataLoad : BOOL;
	bENGCTR_DataLoad : BOOL;
	bMFB50_Dataload : BOOL;
	iIdx : USINT;
	rp49Zyl : ARRAY[0..24] OF REAL;
	bLoad_p49_Map : BOOL;
	ucCylIdx : USINT;
	ucPwrIdx : USINT;
	ucTmpIdx : USINT;
	bOpt_DataLoad : BOOL;
	bAmmSeqClkP : BOOL;
	TON_SecondTick : TON;
	bMapLoaded : ARRAY[0..24] OF BOOL;
	i : INT;
	bMapLoad : BOOL;
	xTON_Reset : TON := (0);
	bPUSL_DataLoad : BOOL := 0;
	bFilt_DataLoad : BOOL := 0;
	bDel_p49_Map : BOOL := 0;
	bWG_DataLoad : BOOL;
	bEG_DataLoad : BOOL;
	bAutoLoad_Ena : BOOL;
	TON_AutoLoad : TON;
	bFS_DataLoad : BOOL;
	bALL_Dataload : BOOL := 0;
	bRKS_DataLoad : BOOL := 0;
	bIG_DataLoad : BOOL := 0;
	bAutoLoad_Ena_TP : BOOL := 0;
	TP_bAutoLoad : TP := (0);
	bSync_DataLoad : BOOL := 0;
	bLX2_DataLoad : BOOL;
	bDAI_DataLoad : BOOL;
	iSA_PIValveType_old : INT; (* old PI valve type to detect value change *)
END_VAR
```

### Program Logical/EngineController/gen_EC_T5 (IEC) - + common tasks @ 100ms

- gen_EC_T5Cyclic.st (not readable text: treated as protected, skipped)

- gen_EC_T5Init.st (not readable text: treated as protected, skipped)

#### gen_EC_T5.var - Local variables
```iecst
(********************************************************************
 * COPYRIGHT -- INNIO Company
 ********************************************************************
 * Program: general_EC
 * File: general_EC.var
 * Author: WaldharM
 * Created: May 22, 2012
 ********************************************************************
 * Local variables of program general_EC
 ********************************************************************)
VAR
	TOF_Act_Release : TOF;
	TON_Act_Mon_Release : TON;
	ucInitIndex : USINT;
END_VAR
```

### Program Logical/EngineController/skip_zde (IEC) - + creating bit pattern to handle a skipfire operation

- skip_zdeCyclic.st (not readable text: treated as protected, skipped)

- skip_zdeInit.st (not readable text: treated as protected, skipped)

#### skip_zde.var - Local variables
```iecst
(********************************************************************
 * COPYRIGHT -- INNIO Company
 ********************************************************************
 * Program: skip_zde
 * File: skip_zde.var
 * Author: Waldharm
 * Created: May 18, 2010
 ********************************************************************
 * Local variables of program skip_zde
 ********************************************************************)
VAR
	bSkipDrehz_O : BOOL; (*interlock bit for overspeed*)
	bSkipDrehz_U : BOOL; (*interlock bit for underspeed*)
	rN_DrehzLeerOben : REAL; (*inner speed level threshold*)
	rN_DrehzLeerUnten : REAL; (*inner speed level threshold*)
	TON_SkipOffset : TON; (*time interval for the misfire rotation*)
	iNum_SkipCyl_Calc_old : USINT; (*store pv for the misfire pattern*)
	rN_InnerThres : REAL; (*inner threshold*)
	iSkip_StartRot : SINT; (*start rotation point*)
	xSigScal_P_Skipfire : xSigScal; (*linear scaling function block*)
	bOnceWM : BOOL; (*rising edge bit*)
	bOnceWM_II : BOOL; (*rising edge bit*)
	usSkipCounter : UINT;
	usCounterLimit : UINT;
	rDivisor_P_Skipfire : REAL;
	xSigScal_FF_Misf : xSigScal;
	xSigScal_FF_Misf2 : xSigScal;
	rN_DownsetSkipfireStart : REAL;
	iNum_SkipCyl_I : SINT;
	iNum_SkipCyl_P : SINT;
	LCCurveByPoints_PMap_Skipfire : LCCurveByPoints;
	refPoint_PMap_Skipfire : ARRAY[0..12] OF lcCurveByPoints_TabEntry_type;
	TOF_SkipState : TOF;
	ucMainOffset : USINT;
	rN_Nom_NReg : REAL;
	rN_NRegOffset : REAL; (*Offset für Leerlaufregler x rpm über Netzfrequenz*)
	FILTER_rSynchFreq : FILTER_R;
	usFreqFiltConst : USINT; (*Filterzeitkonstante [SW-Zyklen] für die Nezufrequenz zur Drehzahlsollwertberechnung*)
	iCnt_NoSkip_HiCtr : SINT;
	iSkip_CylOffs_HiCtr : SINT; (*Hierachie Offset*)
	iCnt_Skip_Cyl : SINT;
	tSkipMisfTOF : TIME;
	rN_Nom_NReg_old : REAL;
	scSkipSyncAdd : SINT; (*frueher global, kommt eventuel irgendwann*)
	i : USINT; (*for statement index*)
	bSkipCyl : ARRAY[0..24] OF BOOL; (*combined Skip pattern*)
	iNum_SkipCyl : SINT; (*additional skipping cylinders to hierachie skipping pattern*)
	iCnt_Rot : USINT; (*Rotation counter*)
	bExCtr_SkipCyl : ARRAY[0..24] OF BOOL;
	bSkipChange : BOOL;
	bSum_SkipCyl : ARRAY[0..24] OF BOOL;
	bSum_SkipCyl_old : ARRAY[0..24] OF BOOL;
	iNum_SkipCylSum : SINT;
	iNum_SkipCylExT : USINT;
	bChangePattern : BOOL;
	iNum_SkipCyl_Calc_old_II : USINT;
	bExCtr_SkipCyl_II : ARRAY[0..24] OF BOOL;
	iNum_SkipCyl_Calc_II : USINT;
	xFSync : fFSync;
	LCRCurveByPoints_SCRTCtr_SkipF : LCRCurveByPoints; (* skip limit for SCR inlet temperature controller over normed power *)
	rSkipF_SCRTCtr : REAL; (* output of SCR inlet temperature controller *)
	rSkipF_SCRTCtr_limited : REAL; (* output of SCR inlet temperature controller limited *)
	bSkipCylActNEW : ARRAY[0..24] OF BOOL;
	xTON_SkipChange : ARRAY[0..24] OF TON; (*Baustein für das verzögerte Abschalten von Zylindern wenn Anzahl der geskippten Zylindern gleich bleibt *) (* Statistic *)
	tiDelaySkipChange : TIME;
	bDelaySkipOFF : BOOL := TRUE; (*Abschalten von Zylindern verzögern wenn Anzahl der geskippten Zylindern gleich bleibt*)
	bSkipCylActOLD : ARRAY[0..24] OF BOOL;
	iNoOfCylExtraCold : INT := 3;
	iNoOfCylExtraWarm : INT := 1;
	rPlim_CylExtra : REAL := 100;
	xF_TRIG_FSyncEnabled : F_TRIG;
END_VAR
```

### Program Logical/EngineController/hum_pac_EC (IEC) - + Humidity Package

- hum_pac.st (not readable text: treated as protected, skipped)

#### hum_pac.var - Local variables
```iecst
(********************************************************************
 * COPYRIGHT -- INNIO Company
 ********************************************************************
 * Program: hum_pac
 * File: hum_pac.var
 * Author: 105051472
 * Created: December 20, 2012
 ********************************************************************
 * Local variables of program hum_pac
 ********************************************************************)
VAR
	TON_SecondTick : TON; (* FUB 1 second timer tick *)
	ssAvgLength : INT; (*[0.1s]*)
	rMixTempDevLimit : REAL; (*[K] oder [°C]*)
	ssMixTempDevCount : INT;
	psatt : REAL;
	ps_LFO : REAL; (*[mbar]*)
	rpl_soll_Max_Sum : REAL;
	rpl_soll_Max_Array : ARRAY[0..2999] OF REAL;
	rpl_ist_Array : ARRAY[0..2999] OF REAL;
	tg_soll_Hum : REAL; (*[°C]*)
	psatt2 : REAL; (* sättigungspartialdruck P red *)
	tg_Hum : REAL; (*[°C]*)
	usCount : UINT;
	usCount2 : INT;
	rpl_ist_Sum : REAL;
	Sim3pCTR_Hum_PRed : Sim3pCTR;
	RT_INFO : RTInfo;
	rCycleTime : REAL; (*[s?]*)
	AbsHumidityCalc : REAL; (* absolute humidity air intake calculated [kg/kg] *)
	AbsHumidityCalc_Mix : REAL; (* absolute humidity mixture calculated [kg/kg] *)
	rpl_soll_Max : REAL;
	xSigScal_Dpl_soll : xSigScal_R;
	tg_soll_HumOffset_corr : REAL; (*correction of charge temperature offset, to keep a control deviation, if in humidity power reduction*)
	rpl_ist : REAL;
	pbaro_p2s : REAL := 1.0; (*p2s Value when engine was stopped the last time (as option in use for humidity control) [bar]*)
	rT_T2_Set_internal : REAL;
	tBM2166Bloc : TIME := T#2m; (*Block B2166 after falling edge*)
	TP_BM2166 : TP;
END_VAR
```

### Program Logical/EngineController/PUSL (IEC) - + power unit safty layer

- PUSLCyclic.st (not readable text: treated as protected, skipped)

- PUSLInit.st (not readable text: treated as protected, skipped)

#### PUSL.var - Local variables
```iecst
(********************************************************************
 * COPYRIGHT -- INNIO Company
 ********************************************************************
 * Program: PUSL
 * File: PUSL.var
 * Author: 502293141
 * Created: April 02, 2014
 ********************************************************************
 * Local variables of program PUSL
 ********************************************************************)
VAR
	bFadOutCyl_Knock : ARRAY[0..24] OF BOOL;
	TON_SecondTick : TON;
	ucCylinderCount : USINT;
	iCnt_TaskCycles : USINT; (*task cycle counter*)
	usLimpHomeCount : ARRAY[0..24] OF UINT;
	usNoLimpHomeCount : ARRAY[0..24] OF UINT;
	bAmmSeqClkP : BOOL;
	HiContrCyl : ARRAY[0..24] OF HiContr;
	bHiCtr_WCCtr_Ena : BOOL;
	bHiCtr_GICtr_Ena : BOOL;
	bHiCtr_PmaxLimCtr_Ena : BOOL;
	ssPmaxLimReachedAnzCyl : INT; (*Anzahl der Zylinder mit PmaxLimReached aus HiContr*)
	rPowRedCyl_HiContrMaxGlob : REAL; (*Max. Leistungsreduktion aus HiContr über alle Zylinder*)
	HiGlobEng : HiGlob;
	bHiGlobEng_EngStopErrAck : BOOL;
	bNO_Pred_HiContr : BOOL; (*TRUE = keine Leistungsreduktion durch Hierarchycontroller*)
	TON_Netp : TON;
	TON_LEANOXON : TON;
	rFehlerFaktor_HiContr : REAL; (*Fehlerfaktor*)
	iNum_Cyl_LimpHome : USINT; (*Anzahl der Zylinder im Limp Home Mode*)
	TON_2287 : TON; (*** modifiziert:*)
	rHiGlobEng_TSkipCount : REAL;
	rHiGlobEng_TSkipCount1 : REAL;
	rHiContrCyl_TGICount : REAL;
	rPr_CPP_AbsLim_old : REAL;
	rP_Set_HiCtr_LimRed : REAL;
	rP_Set_HiCtr_Lim : REAL;
	bHiContrCyl_FaultMFSign : ARRAY[0..24] OF BOOL;
	bHiContrCyl_MFB50Freeze : ARRAY[0..24] OF BOOL;
	bHiContrCyl_OptPIDFreeze : ARRAY[0..24] OF BOOL;
	bHiContrCyl_PmaxLimReached : ARRAY[0..24] OF BOOL;
	rKnck_Intgr_Lim_Hi : REAL;
	rKnck_Intgr_Lim_Lo : REAL;
	iCnt_Cyl_Misf : UINT;
	iCnt_Cyl_Misf2 : UINT;
	iNum_CylPerCycle : USINT; (* execute HiContrCyl for i Cyl per task cycle *)
END_VAR
(* Test Bits *)
VAR
	bTEST_NO_reset : BOOL; (*TRUE = Kein Reset der Testbits*)
	bTEST_kompAussetzer : ARRAY[0..24] OF BOOL;
	bTEST_Aussetzer : ARRAY[0..24] OF BOOL;
	bTEST_Misf_II : ARRAY[0..24] OF BOOL;
	bTEST_GluehZuend : ARRAY[0..24] OF BOOL;
	bTEST_FaultMFSign : ARRAY[0..24] OF BOOL;
	bTEST_MFB50Freeze : ARRAY[0..24] OF BOOL;
	bTEST_OptPIDFreeze : ARRAY[0..24] OF BOOL;
	bTEST_PmaxLimReached : ARRAY[0..24] OF BOOL;
	bTEST_SkipCyl : ARRAY[0..24] OF BOOL;
	bLimpHome_TestBit : ARRAY[0..24] OF BOOL;
END_VAR
(* Perm Parameters *)
VAR
	TON_misf_start : ARRAY[0..24] OF TON;
	TON_misf_trip : ARRAY[0..24] OF TON;
	ti_OpTi_MisfCyl_old : TIME;
	bHiContrACTIVE : BOOL;
	LCRCByP_TupMFshape : LCRCurveByPoints;
	rCorrLeanox_Rise : REAL;
	rCorrLeanox_Sink : REAL;
	RAMPE_R_LeanoxCorr : RAMPE_R;
	i : USINT;
	bTEST_bLimpHome : ARRAY[0..24] OF BOOL;
	bLimpHomeCylWarn : ARRAY[0..24] OF BOOL;
	ucNoOfCylFailAll : USINT;
	LCRCByP_NoOfFailAll : LCRCurveByPoints;
	bFreezeOptiAll : BOOL;
	bOM_InfoMisf : ARRAY[0..24] OF BOOL;
	iCnt_Misfire : ARRAY[0..24] OF UINT;
	iNum_Cyl_MaxMisf : UINT;
	iNum_Misf_Cycles : UINT;
	LCRCByP_P2s_MisfCycles : LCRCurveByPoints;
	LCRCByP_P2s_MisfMaxCyl : LCRCurveByPoints;
	LCRCByP_MaxCylSkipBefStop : LCRCurveByPoints;
	refPoint_MaxCylSkipBefStop : ARRAY[0..1] OF lcrCurveByPoints_TabEntry_type;
END_VAR
```

### Program Logical/EngineController/pi_bal_EC (IEC) - + cylinder balancing with port injection

- pi_balCyclic.st (not readable text: treated as protected, skipped)

- pi_balInit.st (not readable text: treated as protected, skipped)

#### pi_bal.var - Local variables
```iecst
(********************************************************************
 * COPYRIGHT -- INNIO Company
 ********************************************************************
 * Program: pi_bal
 * File: pi_bal.var
 * Author: WaldharM
 * Created: December 11, 2009
 ********************************************************************
 * Local variables of program pi_bal
 ********************************************************************)
VAR
	RFILTER_Pmax : ARRAY[0..24] OF FILTER_R;
	RMEDIAN24_Pmax : RMEDIAN24;
	ucBalAvgCounter : USINT;
	LCRPIDpara_Bal : ARRAY[0..24] OF LCRPIDpara;
	LCRPID_Bal : ARRAY[0..24] OF LCRPID;
	rDeadbandBalancing : REAL;
	ucSampleRate : USINT;
	usCycleTime : UINT;
	bMapSave : BOOL;
	rDur_Sum_Avg : REAL;
	rDur_Map : ARRAY[0..24] OF REAL;
	TON_BalSafetyStop : TON;
	LIndex : USINT;
	x1y1 : REAL;
	x2y1 : REAL;
	x2y2 : REAL;
	x1y2 : REAL;
	x1Wert : REAL;
	x2Wert : REAL;
	rLoQuanti_P_Dev : REAL;
	rUpQuanti_P_Dev : REAL;
	rLoQuanti_T_Dev : REAL;
	rUpQuanti_T_Dev : REAL;
	bExitExit : BOOL;
	rZM : REAL;
	bKennfelderauslesen : BOOL;
	bManual_Bal : BOOL;
	bBal_TimeOut : BOOL;
	xLCRCbyP_KpMap_PID1 : LCRCurveByPoints;
	xLCRCbyP_KpMap_PID2 : LCRCurveByPoints;
	RFILTER_Pmax_PID2 : ARRAY[0..24] OF FILTER_R;
	LCRLimScal_BalCritOn : LCRLimScal;
	LCRLimScal_BalCritOff : LCRLimScal;
	TON_SS_P2s : TON;
	rP2s_Ref : REAL;
	TON_SS_T2s : TON;
	rT2s_Ref : REAL;
	TON_Kennfeldauslesen : TON;
	TON_SS_Pel : TON;
	rPel_Ref : REAL;
	rLimpHomeDownset : REAL;
	rPMaxOffset_raw : ARRAY[0..24] OF REAL;
	rPMaxOffset_raw_2 : ARRAY[0..24] OF REAL;
	x1y1_P49 : REAL;
	x1y2_P49 : REAL;
	x2y1_P49 : REAL;
	x2y2_P49 : REAL;
	x1Wert_P49 : REAL;
	x2Wert_P49 : REAL;
	rP_D_p49_Map : ARRAY[0..24] OF REAL;
	rP_D_p49_Measure : ARRAY[0..24] OF REAL;
	rZM_DP49 : ARRAY[0..24] OF REAL;
	rPMaxOffset_raw_3 : ARRAY[0..24] OF REAL;
	rPMaxOffset_limit : ARRAY[0..24] OF REAL;
	rSumCor_rPMaxOffset : REAL;
	RMEDIAN24_p49 : RMEDIAN24;
	RMEDIAN24_IHR : RMEDIAN24;
	RFILTER_P49 : ARRAY[0..24] OF FILTER_R;
	RFILTER_IHR	: ARRAY[0..24] OF FILTER_R;
	rPMaxOffset_bar : ARRAY[0..24] OF REAL;
	bBalRequired_Arr : ARRAY[0..24] OF BOOL;
	bPID_Init : BOOL;
	ucBal_State_Old : USINT;
	rDur_Sum : REAL;
	bReleaseBalancing : BOOL;
	ucBal_State : USINT;
	bBalRequired : BOOL;
	rPmax_Filter : ARRAY[0..24] OF REAL;
	rPmax_Filter_Avg : REAL;
	rNNet_NPoint_Quanti : REAL;
	rPMaxOffset : ARRAY[0..24] OF REAL;
	iIdx_T2s_ReC : USINT;
	iIdx_P2s_Loop : USINT;
	iIdx_T2s_Loop : USINT;
	iIdx_T2s_Loop_Inv : USINT;
	iIdx_T2s_MapSize : USINT;
	iIdx_T2s : USINT;
	iIdx_P2s_MapSize : USINT;
	iIdx_P2s : USINT;
	iIdx_P2s_ReC : USINT;
	iIdx_Cyl : USINT; (*Zylinder Zähler*)
	rCA_Dur_Lim_Lo : REAL;
	rCA_Dur_Lim_Hi : REAL;
	bMapSave_p49 : BOOL; (*Alt: bSW6*)
	iIdx_Pr : USINT;
	iIdx_T : USINT;
	iCycle : USINT;
	fub_RTInfo : RTInfo;
	bTrigger : BOOL;
	TP_MapSave : TP;
	bOptRel : BOOL;
	rPr_P49_Avg : REAL;
	rPr_PMax_SumCor : REAL;
	rP49_Filter : ARRAY[0..24] OF REAL;
	RFILTER_P49_PID2 : ARRAY[0..24] OF FILTER_R;
	bDur_Lim_PID2 : ARRAY[0..24] OF BOOL;
	bDur_Lim_PID2_Warn : ARRAY[0..24] OF BOOL;
	rCA_PI_Dur_SOffset_raw : ARRAY[0..24] OF REAL;
	TON_SecondTick : TON;
	bAmmSeqClkP : BOOL;
	bMapSave_Ena : BOOL;
	rPmaxOffset_UL : REAL;
	rPmaxOffset_LL : REAL;
	rPmax_Offset_Coef_a : REAL;
	rPmax_Offset_Coef_b : REAL;
	rLim_PID2_Hi : REAL;
	rLim_PID2_Lo : REAL;
	xTP_ResetMap : TP;
	xTP_CommModeOn : TP;
	xTP_CommModeOff : TP;
	xTP_SaveToMap : TP;
	bP49_Source : BOOL;
	bTEST_NEW_SS : BOOL;
	rPmax_Offset_Coef_d : REAL;
	xLCRCByP_d_P2s : LCRCurveByPoints;
	rPmax_Offset_Coef_e : REAL;
	rPID_e : REAL;
	rPID_e_cyl : REAL;
	xMEDIAN_MFBvar : RMEDIAN24;
	xFILTER_MFBvar : ARRAY[0..24] OF FILTER_R;
	rCA_MFBvar_dlt_Filt : ARRAY[0..24] OF REAL;
	rPmax_Offset_Coef_b_IP : REAL;
	xFILTER_IP : ARRAY[0..24] OF FILTER_R;
	rPMaxOffset_raw_1 : ARRAY[0..24] OF REAL;
	xLCRCByP_c_P2s : LCRCurveByPoints;
	xLCRCByP_e_P2s : LCRCurveByPoints;
	rPmax_Offset_d_lim : ARRAY[0..24] OF REAL;
	rPmax_Offset_c : ARRAY[0..24] OF REAL;
	rPmax_Offset_d : ARRAY[0..24] OF REAL;
	rPmax_Offset_Coef_c : REAL;
	bLockCommissioning : BOOL; (*Lock commissioning and map saving if in G2 mode*)
	bLockCommissioning_FAR : BOOL; (*Lock commissioning and map saving if FAR out of bound*)
	bFAR_lim_lock_Comm : ARRAY[0..24] OF BOOL; (*Lock commissioning because FAR is out of bound *)
	xTOF_FAR_lim_comm_blocked : ARRAY[0..24] OF TOF; (*TOF for comissioning blocked because FAR is out of bound *)
	bFAR_lim_comm_blocked : ARRAY[0..24] OF BOOL; (*comissioning blocked because FAR is out of bound *)
	TON_OptiCyl_Lim : ARRAY[0..24] OF TON;
	x1 : REAL := 0.0;
	x2 : REAL := 0.0;
	y1 : REAL := 0.0;
	y2 : REAL := 0.0;
	xTOF_bLimpHomeCyl : ARRAY[0..24] OF TOF;
	tiDel_TOF_LimpHome : TIME := T#10s;
	rDownSetTOF_LH : REAL := -2;
	bDur_Opt_Lim : ARRAY[0..24] OF BOOL;
	bDur_Opt_Lim_Warn : ARRAY[0..24] OF BOOL;
	xTON_Opt_Dur_Lim : ARRAY[0..24] OF TON;
	tiLim_Dur_Off : TIME; (* Time delay before Duration Offset Limitation Warning is triggered *)
	rCA_Lim_Dur_Margin : REAL; (* Margin to limit to trigger offset duration limitation Warning *)
	rQuantifier_Opt_Gauss : REAL; (* Quantifier for gauss distriburtion *)
	rSigma_Opt_p2s : REAL; (* sigma for gauss distribution in charge pressure direction *)
	rSigma_Opt_T2s : REAL; (* sigma for gauss distribution in charge temperature direction *)
	xGR_MAXR_Opt_Req_CL : GR_MAXR := (0); (*hysterisis for PID ouput to request automatic balancing *)
	xTON_Opt_Req_CL : TON; (* delay for request automatic balancing *)
	xTON_Opt_Done : TON; (* delay for request automatic balancing *)
	bOpt_Req_CL : BOOL; (* request automatic balancing *)
	rDur_Off_CL_max : REAL; (* maximum of all PID outputs for cylinder balancing *)
	rIHR_set : ARRAY[0..24] OF REAL;
	rFAR_set : ARRAY[0..24] OF REAL;
	rFAR_act : ARRAY[0..24] OF REAL;
	bFAR_up_lim : ARRAY[0..24] OF BOOL;
	bFAR_low_lim : ARRAY[0..24] OF BOOL;
	rK_Opt_a_fact : REAL; (* k factor for linear interpolation of a-Factor on IHR *)
	rD_Opt_a_fact : REAL; (* d offset for linear interpolation of a-Factor on IHR *)
END_VAR
```

### Program Logical/EngineController/pi_ctr_EC (IEC) - + controller for the port injection valve

- pi_ctrCyclic.st (not readable text: treated as protected, skipped)

- pi_ctrInit.st (not readable text: treated as protected, skipped)

#### pi_ctr.typ
```iecst
(********************************************************************
 * COPYRIGHT -- INNIO Company
 ********************************************************************
 * Program: pi_ctr
 * File: pi_ctr.typ
 * Author: WaldharM
 * Created: August 06, 2010
 ********************************************************************
 * Local data types of program pi_simu
 ********************************************************************)

TYPE
	lcCurveByPoints_REAL_TbEtry_type : 	STRUCT
		x : REAL;
		y : REAL;
	END_STRUCT;
END_TYPE
```

#### pi_ctr.var
```iecst
(********************************************************************
 * COPYRIGHT -- INNIO Company
 ********************************************************************
 * Program: pi_ctr
 * File: pi_ctr.var
 * Author: WaldharM
 * Created: February 13, 2009
 ********************************************************************
 * Local variables of program pi_ctr
 ********************************************************************)
VAR
	rQg_set_B : REAL; (*volumetric flow rate bank B*)
	rQg_set_A : REAL; (*volumetric flow rate bank A*)
	bAmmSeqClkP : BOOL; (*trigger for AMM_Sequence*)
	rHub : REAL; (*stroke [dm]*)
	rSpezGasd : REAL; (*specific gas density*)
	rEDKappaME : REAL; (*ratio of specific heat*)
	rKappaDKappaPE : REAL; (*ratio of specific heat*)
	rKappaDKappaME : REAL; (*ratio of specific heat*)
	rZDKappa : REAL; (*ratio of specific heat*)
	rKappaPEDKappa : REAL; (*ratio of specific heat*)
	rKappaBruch : REAL; (*ratio of specific heat*)
	rZDKappaPE : REAL; (*ratio of specific heat*)
	rTventil_B : REAL; (*opening time bank B [sec.]*)
	rCAv_B : REAL; (*opening time bank B [°CA]*)
	rTventil_A : REAL; (*opening time bank A [sec.]*)
	rCAv_A : REAL; (*opening time bank A [°CA] *)
	rQg_Zaehler_B : REAL; (*numerator bank B  (gas amount per cylinder)*)
	rQg_Zaehler_A : REAL; (*numerator bank A  (gas amount per cylinder)*)
	rQm_ventil : REAL; (*mass flow rate per second for the valve*)
	rZM200 : REAL; (*intermediate memory*)
	rZM206 : REAL; (*intermediate memory*)
	rZM205 : REAL; (*intermediate memory*)
	rZM202 : REAL; (*intermediate memory*)
	rZM201 : REAL; (*intermediate memory*)
	rZM204 : REAL; (*intermediate memory*)
	rQg_Nenner_B : REAL; (*denominator bank B (gas amount per cylinder)*)
	rQg_Nenner_A : REAL; (*denominator bank A (gas amount per cylinder)*)
	rBohr : REAL; (*bore diameter [dm]*)
	ulUnivPos : ARRAY[0..24] OF UDINT;
	TON_SecondTick : TON;
	ucSAFINr : USINT;
	bPIDuration_HIGH : ARRAY[0..24] OF BOOL;
	RAMPE_Lambda : RAMPE_R;
	rDurGradLimit : REAL;
	rCAv_A_LastCycle : REAL;
	rCAv_B_LastCycle : REAL;
	rGrid_Offset : REAL;
	PiDurMapIndex : INT;
	ucPiDur_X1 : INT;
	ucPiDur_X2 : INT;
	rDp_Gasrail : REAL;
	ucDp_GR_Y1 : INT;
	ucDp_GR_Y2 : INT;
	x1y1 : REAL;
	x1y2 : REAL;
	x2y1 : REAL;
	x2y2 : REAL;
	x1Wert : REAL;
	x2Wert : REAL;
	rCorr_PI_Dur : REAL;
	rCA_PI_Timing : REAL;
	rHubVolumen : REAL;
	rQm_set_A : REAL;
	rQm_set_B : REAL;
	bPIDurationFix_Act : BOOL;
	rCA_Dur_L : ARRAY[0..12] OF REAL;
	rCA_Dur_H : ARRAY[0..12] OF REAL;
	rCA_Dur_Fix : REAL;
	LCRCByP_ZWert : LCRCurveByPoints;
	r_ZWert_scal : REAL;
	bPortInject_Rel : BOOL;
	rPr_P2s_limit_LamMisf : REAL;
	LCRCByP_LambdaRamp : LCRCurveByPoints;
	tLambdaRampMap : ARRAY[0..9] OF lcrCurveByPoints_TabEntry_type;
	iCyl : USINT;
	TP_PI_Block : TP;
	rTi_PI_Duration : REAL;
	bLamLim : BOOL;
	xTOF_LamLim : TOF := (0);
	bPI_Block : ARRAY[0..24] OF BOOL;
	xTON_GR_Scav : TON := (0);
	bGR_Scav : BOOL;
	xRAMPE_Pr_Signal : RAMPE_R;
	rDurGradLimitIsland : REAL;
	iTFilt_p2s_des : UINT := 50;
	xFILTER_R_p2s_des : FILTER_R;
	rPr_p2sSet_Limit4Fast_Signals : REAL := 0.2;
	rPr_p2sSet_LamLimLoadAcc : REAL := 0.2; (* 0.55 *)
	tiLambdaLoadAcc : TIME := T#1200ms;
	rPr_p2sSet_LamLimLoadRej : REAL := 10;
	tiLambdaLoadRej : TIME := T#600ms;
	xTP_LoadAcc : TP;
	xTP_LoadRej : TP;
	xTON_MaxTime : TON := (0);
	bLamDelta_run : BOOL;
	tiMaxDuration : TIME := T#1500ms;
	xTON_DeltaLam_Off : TON := (0);
	bBlock_LamDelta : BOOL := 0;
	rN_LimitSS : REAL := 15;
	tiDelaySS : TIME := T#2s;
	xTON_N_SS : TON;
	ParaEC_rHCR_Max1 : REAL;
	bGR_Scav_H : BOOL; (* activates gas rail scavanging for additional cylinders *)
	iCA_Dur_Max : UINT; (* defines maximum opening duration of pi 10x°CA *)
	xDTGetTime : DTGetTime;	(* Timer for engine standstill *)
	DT_Eng_Stop : DATE_AND_TIME; (* Date and time when engine was stopped *)
	rCA_GR_Scav : REAL;	(*Gas rail scavanging CA duration*)
	rLambda_Min : REAL;	(*Lambda minimum*)
	iNum_Cyl_Plausible : INT; (* amount of plausible cylinders for the Lambda PBC calculation  *)
	rIHR_Sum : REAL; (* Sum of the integral heat release values for the mean value calculation *)
	rPr_49bfTDC_Sum : REAL; (* Sum of the P49bfTDC values for the mean value calculation *)
	rIHR_Mean : REAL; (* mean value of the integral heat release values for the mean value calculation *)
	rPr_49bfTDC_Mean : REAL; (* mean value of the P49bfTDC values for the mean value calculation *)
	xRMEDIAN24_P49 : RMEDIAN24; (* Median of the P49bfTDC for the plausibility check for the Lambda PBC calculation *)
	xRMEDIAN24_IHR : RMEDIAN24; (* Median of the IHR for the plausibility check for the Lambda PBC calculation *)
	rFAR_Lam_PBC : REAL; (* fuel to air ratio for the lambda PBC calculation*)
	iIdx_Cyl : USINT; (* cylinder counter *)
	rIHR_buf : ARRAY[0 .. 24] OF REAL; (* IHR buffer for median calculation *)
	iNum_IHR_buf : USINT; (* size of IHR buffer for median calculation *)
	xLamCtrPBC : fLamCtrPBC; (* lambda controller for port injection *)
	rLam_PBC_unfilt : REAL; (* unfiltered lambda calculated from in-cylinder data *)
	xFILTER_Lam_LamCtrPBC : FILTER_R; (* filter for lambda controller PBC *)
	bLamCtrPBC_freeze : BOOL; (* freeze lambda controller PBC in case of bad lambda estimation *)
	ru_LamCtrPBC_freeze : REAL; (* freezed output value for lambda controller PBC *)
	xTOF_bLamCtrPBC_freeze : TOF; (* delay of lambda freeze bit *)
END_VAR
```

### Program Logical/EngineController/psi_cal (IEC) - + calculates stoich. power

- psi_cal.st (not readable text: treated as protected, skipped)

#### psi_cal.var - Local variables
```iecst
(********************************************************************
 * COPYRIGHT -- INNIO Company
 ********************************************************************
 * Program: psi_cal
 * File: psi_cal.var
 * Author: WaldharM
 * Created: December 03, 2012
 ********************************************************************
 * Local variables of program psi_cal
 ********************************************************************)
VAR
	LCRCByP_Eta_Eng : LCRCurveByPoints;
	rEta_Eng : REAL;
	LCRCByP_Eta_Gen : LCRCurveByPoints;
	rEta_Gen : REAL;
END_VAR
```

### Program Logical/EngineController/SPP_TC1 (IEC) - + provides global IO Data

- SPP_TC.st (not readable text: treated as protected, skipped)

#### SPP_TC.var - Local variables
```iecst
(********************************************************************
 * COPYRIGHT -- INNIO Company
 ********************************************************************
 * Program: SPP_EC
 * File: SPP_EC.var
 * Author: 502293141
 * Created: March 20, 2014
 ********************************************************************
 * Local variables of program IOScal_EC
 ********************************************************************)
VAR
	iIdx_Filt_Cycles : UINT;
	xFilter_R_P2s : FILTER_R;
	xFilter_R_P2s_B : FILTER_R;
	xFilter_R_P2s_A : FILTER_R;
	xFilter_R_P2s_Avg : FILTER_R;
	xFilter_R_Pr_DAI_A : FILTER_R;
	xFilter_R_Pr_DAI_B : FILTER_R;
	xFilter_R_Pr_DAI_In : FILTER_R;
	xFilter_R_T_DAI : FILTER_R;
	xFilter_R_P1 : FILTER_R;
	xFilter_R_P1_A : FILTER_R;
	xFilter_R_P1_B : FILTER_R;
	xFilter_R_P1_Avg : FILTER_R;
	xFilter_R_Pr_EGbHPTC_A : FILTER_R;
	xFilter_R_Pr_EGbHPTC_B : FILTER_R;
	xFilter_R_Pr_EGbHPTC_Avg : FILTER_R;
	xFilter_R_Pr_EGaHPTC_A : FILTER_R;
	xFilter_R_Pr_EGaHPTC_B : FILTER_R;
	xFilter_R_Pr_EGaHPTC_Avg : FILTER_R;
	xFilter_R_Pr_EGaLPTC_A : FILTER_R;
	xFilter_R_Pr_EGaLPTC_B : FILTER_R;
	xFilter_R_Pr_EGaLPTC_Avg : FILTER_R;
	xFilter_R_GR : FILTER_R;
	status : UINT := 0;
	tRTC_FirstTC1InitStart : rtctime_typ := (0);
END_VAR
```

### Program Logical/EngineController/SPP_EC (IEC) - + provides global IO Data

- SPP_EC.st (not readable text: treated as protected, skipped)

#### SPP_EC.var - Local variables
```iecst
(********************************************************************
 * COPYRIGHT -- INNIO Company
 ********************************************************************
 * Program: SPP_EC
 * File: SPP_EC.var
 * Author: 502293141
 * Created: March 20, 2014
 ********************************************************************
 * Local variables of program IOScal_EC
 ********************************************************************)
VAR
	LCRMovAvg_rPr_GR_fast : LCRMovAvgFlt;
	LCRMovAvg_rPr_GR : LCRMovAvgFlt;
	LCRMovAvg_rPr_P2s_fast : LCRMovAvgFlt;
	LCRMovAvg_rPr_P2s : LCRMovAvgFlt;
	LCRMovAvg_rPr_P2s_A : LCRMovAvgFlt;
	LCRMovAvg_rPr_P2s_B : LCRMovAvgFlt;
	iIdx_Cyl : USINT;
	DTGetTime_RPS : DTGetTime;
	LCRMovAvg_rPr_P2s_Opt : LCRMovAvgFlt;
	iFilt_fast : UINT := 3;
	iFilt : UINT;
	iFilt_Old : UINT;
	iFilt_Opt : UINT;
	iFilt_Opt_Old : UINT;
	iSort_Cache : USINT;
	xFilter_R_T_SCR_In : FILTER_R; (* Filter for SCR inlet temperature controller input *)
END_VAR
```

### Program Logical/EngineController/gassort_int (IEC) - + provides data for gassort 0

- gassort_intCyclic.st (not readable text: treated as protected, skipped)

#### gassort_int.var - Local variables
```iecst
(********************************************************************
 * COPYRIGHT -- INNIO Company
 ********************************************************************
 * Program: gassort_int
 * File: gassort_int.var
 * Author: Caks
 * Created: Aug 06, 2014
 ********************************************************************
 * Local variables of program gassort_int
 ********************************************************************)
VAR
	iIdx_loop : INT;
	rCA_IgnP_Offs_H2_Prior : REAL; (* ITP offset via H2 content before H2 switching point [degCA] *)
	rCA_IgnP_Offs_H2_After : REAL; (* ITP offset via H2 content after H2 switching point [degCA] *)
	rLHV_H2 : REAL := 2.997; (* Lower heating value Hydrogen [kWh/m3] *)
	rStdGD_H2 : REAL := 0.089; (* Standard gas density Hydrogen [kg/m3] *)
	rMinAirReq_H2 : REAL := 1.972; (* Minimum air requirement Hydrogen [l/l] *)
	rHCR_H2_Comp : REAL := 1.405; (* Heat capacity ratio *)
	rLam_Start_Offset_H2 : REAL; (* Actual calculated start lambda offset depending on H2 content *)
END_VAR
```

### Program Logical/EngineController/PBC (IEC) - + handle the monitoring part for the pressure based control

- PBC.st (not readable text: treated as protected, skipped)

#### PBC.var
```iecst
(********************************************************************
 * COPYRIGHT -- INNIO Company
 ********************************************************************
 * Program: pbc_mon
 * File: pbc_mon.var
 * Author: WaldharM
 * Created: September 15, 2009
 ********************************************************************
 * Local variables of program pbc_mon
 ********************************************************************)
VAR
	AmmSeq_PiCountPosAbw : AmmSequence; (* Trip: Axxxx, OM: Bxxxx, *) (* Oldname: AmmSeq_PiCountPosAbw *)
	AmmSeq_PiNegAbw : AmmSequence; (* Trip: A2275, OM: B2849, Misfiring failure PBC*) (* Oldname: AmmSeq_PiNegAbw *)
	bAmmSeqClkP : BOOL;
	TON_SecondTick : TON;
	bAussetzerTest : BOOL;
	usMinCounter : UINT;
	ssZeitBasisAussetzer : INT;
	ucCylIndex : USINT; (*Schleifenindex*)
	xTOF_PBC : TOF;
	iMotorCycle : INT;
	TOF_P2s : TOF;
	iCnt_IMEP_Misf_sum : USINT;
	iCnt_IMEP_Misf : ARRAY[0..24] OF USINT;
	bCnt_IMEP_Misf : ARRAY[0..24] OF BOOL;
	bCnt_IMEP_NegDev : ARRAY[0..24] OF BOOL; (* Oldname: bPiNegAbw *)
	bCnt_IMEP_PosDev : ARRAY[0..24] OF BOOL; (* Oldname: bPiPosAbw *)
	iCnt_IMEP_NegDev : ARRAY[0..24] OF INT; (* Oldname: ucCountPiNegAbw *)
	iCnt_IMEP_PosDev : ARRAY[0..24] OF INT; (* Oldname: ucCountPiPosAbw *)
	xTP_IMEP_MisfCnt : TP;
	bCPP_AbsLim : ARRAY[0..24] OF BOOL; (* CPP Integrator maximal cylinder pressure absolute limit reached *)
	iCnt_CPP_DevLim : ARRAY[0..24] OF INT; (*Zähler der Überscheitungen des Spitzendrucklimits*) (* Oldname: ucCountPmaxLimit *)
	iCnt_CPP_DevLimOK : ARRAY[0..24] OF INT; (* Zähler der Unterschreitungen des Spitzendruckslimits*) (* Oldname: ucCountPmaxLimitKehr *)
	bRel_CPP_DevLim : BOOL; (* Oldname: bFGAmmSeq_PmaxLimit *)
	xTP_Rel_CPP_DevLim : TP; (* Oldname: TP_FGammSeq_Pmax *)
	bCPP_Warning : ARRAY[0..24] OF BOOL;
	bRel_CPP_AbsLim_W : BOOL; (* Oldname: bFGAmmSeq_PmaxLimit_W *)
	xTP_Rel_CPP_AbsLim_W : TP; (* Oldname: TP_FGammSeq_Pmax_W *)
	bPBC_MSST : BOOL;
	iCnt_IPC_MSF : INT;
	iCnt_PBC_MSF_Delay : ARRAY[0..24] OF INT;
	bPBC_CPP_MSF : ARRAY[0..24] OF BOOL;
	iIdx_Cyl_Act : INT;
	iIdx_MBFvar : INT;
	xTON_MisfPos : TON;
	iCnt_Misf_II : ARRAY[0..24] OF DINT;
	xTON_exec_CQ : TON;
	tCQ : TIME := T#10s; (*Zeitschritte für CQ Ermittlung (Combustion Quality)*)
	iCyl : USINT;
	rNcqCyl : REAL;
	rCQnCyl : ARRAY[0..24] OF REAL;
	rCQnMaxCyl : ARRAY[0..24] OF REAL;
	bCQnMaxReset : BOOL;
	xCppInt : ARRAY[0..24] OF fCPP_Int; (* Cylinder Pressure Peak Limit Integrator *)
	bReset_CPP_LimEvent : BOOL; (* Reset CPP limit counter *)
	xR_TRIG_CppInt_IPRed : ARRAY[0..24] OF R_TRIG; (* Rising Edge - CPP Integrator Ignition Point reduction *)
	bCppInt_IPRed_Trig : ARRAY[0..24] OF BOOL; (* CPP Integrator Ignition Point reduction Operation Message Logged trigger *)
	iCnt_CppInt_IntLimHi : USINT; (* Cylinder Count at CPP Integrator Level Limit High *)
	xTON_CPPInt_IPRed_Off : ARRAY[0..24] OF TON; (* delay for deactivating operating message 2960 *)
	bCppInt_IPRed : BOOL; (* Bit to enable OM block for IT retard from CPPInt *)
END_VAR
```

### Package Logical/EngineController/Sondergas - new EC

### Program Logical/EngineController/Sondergas/SGas (IEC, version 4.07.1) - + Sondergasfunktionen

- SGasCyclic.st (not readable text: treated as protected, skipped)

- SGasInit.st (not readable text: treated as protected, skipped)

#### SGas.var - Local variables
```iecst
(********************************************************************
 * COPYRIGHT -- INNIO Company
 ********************************************************************
 * Program: SGas
 * File: SGas.var
 * Author: 502650054
 * Created: August 19, 2016
 ********************************************************************
 * Local variables of program SGas
 ********************************************************************)
VAR
	iCyl : INT;
	iTaskCycleCOUNT : INT;
	rMFB50Ctr_umax : REAL;
	rMFB50Ctr_umin : REAL;
	rMFB50top2s_kp : REAL;
	rMFB50top2s_ki : REAL;
	rMFB50Ctr_MFB50_max : REAL;
	rMFB50Ctr_MFB50_min : REAL;
	rMFB50Ctr_kp : REAL;
	rMFB50Ctr_ki : REAL;
	rMFB50Ctr_Kt : REAL;
	rMFB50Ctr_T_filt_MFB50 : REAL;
	rMFB50Ctr_MFB50ref : REAL;
	bMFB50Ctr_ON : BOOL;
	iMFB50top2s_mode : INT;
	rMFB50top2s_uman : REAL;
	rMFB50errmax : REAL;
	rMFB50errmin : REAL;
	rMFB50erravg : REAL;
	rITsatmax : REAL;
	rITsatmin : REAL;
	xMEDIAN24_MFB50err : RMEDIAN24;
	xMEDIAN24_Umsatz : RMEDIAN24;
	rUmsatzMEDIAN : REAL;
	CoV_fun : CoV;
	xMEDIAN24_CoV : RMEDIAN24;
	LCRLimScal_umin : LCRLimScal;
	LCRLimScal_umax : LCRLimScal;
	SimPID4_CoV : SimPID4;
	rCoV_Set : REAL;
	rPr_p2s_Range : REAL; (*[bar]*)
	bCoVCtr_act : BOOL;
	rTB34_Set : REAL;
	rTB34_min : REAL;
	rTB34Ctr_kp : REAL;
	rTB34Ctr_ki : REAL;
	SimPID4_TB34 : SimPID4;
	LCRLimScal_MFB50ref : LCRLimScal;
	LCRLimScal_CoVref : LCRLimScal := (0);
END_VAR
```

### Program Logical/EngineController/Sondergas/GlowIGN (IEC) - + formerly known as robits_1 & 2

- GlowIGNCyclic.st (not readable text: treated as protected, skipped)

- GlowIGNInit.st (not readable text: treated as protected, skipped)

#### GlowIGN.var - Local variables
```iecst
VAR
	bFPR_Timer : BOOL; (* fix valves delay time is running *)
	bSCO_Timer : BOOL; (* fix valves delay time is running *)
	bSCO_PBC_Req : BOOL; (*Sicherheitsschliessen angefordert, DMR*)
	xTP_SCO_1 : TP;
	xTON_SCO_2 : TON;
	xTP_SCO_2 : TP;
	xTOF_SCO : TOF;
	FA_TS_UW : GR_MINR;
	i : USINT; (* Counter variable *)
	bSCO_Rel_1 : BOOL := 0; (* Sicherheitsschliessen Gasventil 1 *)
	bSCO_Rel_2 : BOOL := 0; (* Sicherheitsschliessen Gasventil 2 *)
	xTON_FPR : TON; (* delay time for fix valves PRED *)
	xTON_SCO : TON; (* delay time for fix valves VALVE *)
	xTP_FPR_block : TP;
	xTP_SCO_block : TP;
	bSCO_EGT_DevLim : BOOL;
	bSCO_PBC_Rel : BOOL; (*Auslösen Sicherheitsschließen DMR*)
	bSCO_Ena : BOOL; (*Sicherheitsschließen freigegeben*)
	rLam_old : REAL;
	bFPR_LimMax : BOOL; (* Leistungsreduktion wegen maximaler anzahl an FPR*) (* Oldname: bmaxPRed; *)
	rPr_Error : REAL;
	bLeanox_Man_old : BOOL;
	xLCRPT1_FA_GMISCH : LCRPT1;
	bSCO_Rel : BOOL; (*safety cut out release*)
	xTON_30min : TON;
	bEngBlock : BOOL;
	xTP_BLOCK : TP;
	bSCO_Ena_2 : BOOL; (*Freigabe Schliessen Gasventil 2*)
	xCnt_FPR_Max : COUNTER50;
	xTP_2 : TP;
	xCnt_Block1 : COUNTER100;
	xCnt_Block2 : COUNTER100;
	iCnt_100ms : INT;
	rPLevel1 : REAL;
	rPLevel2 : REAL;
	rP_Act_Norm_Filt_OLD3 : REAL;
	rP_Act_Norm_OLD1 : REAL;
	rP_Act_Norm_OLD2 : REAL;
	rP_Act_Norm_Filt_OLD2 : REAL;
	rP_Act_Norm_Filt_OLD1 : REAL;
	bBackFireNetP : BOOL;
	Ring_P2sMon : RING500_R;
	Ring_PowMon : RING1000_R;
	bSG_P2s_GlowRed : BOOL;
	bSG_Pow_GlowRed : BOOL;
	bSG_GlowRed : BOOL;
	xTOF_Block2 : TOF;
	rPr_IMEP_sum : REAL;
	rIMEPLevel1 : REAL;
	rIMEPLevel2 : REAL;
	rPr_IMEP_sum_OLD1 : REAL;
	rPr_IMEP_sum_OLD2 : REAL;
	bBackFirePBC : BOOL;
	rPos_Gm_old : REAL;
	bGlowIGN_Off : BOOL; (* Deactivate Glow ignition detection *)
	bLeanox_Man_old_FGQC : BOOL; (* LEANOX status before FGQC *)
	rLam_old_FGQC : REAL; (* Lambda setpoint before FGQC *)
	rPos_Gm_old_FGQC : REAL; (* Gas mixer setpoint before FGQC *)
	xTP_T1_FGQC : TP; (* Delay time after customer signal *)
	xTP_T2_FGQC : TP; (* Deactivated glow ignition detection *)
	xTP_T3_FGQC : TP; (* Freeze of Controller *)
	xTP_T4_FGQC : TP; (* Delay until function can be activated again *)
	rPos_FGQC_TV : REAL; (* Actual position of TV *)
	rPos_FGQC_CBV : REAL; (* Actual position of CBV *)
	tiGasQualChange_Release : TIME; (* Delay time until function can be activated again *)
END_VAR
```

### Library Logical/EngineController/Sondergas/lAI50toIT (ANSIC, version 2.00.0)

#### lAI50toIT.fun
```iecst
FUNCTION_BLOCK AI50toIT
  VAR_INPUT
    ssMethodType: SINT;
  END_VAR  VAR_INPUT
        mode : INT := 3; (**)
  END_VAR
  VAR_INPUT
        reset : BOOL := FALSE; (**)
  END_VAR
  VAR_INPUT
        umin : REAL := -3.0000000000; (**)
  END_VAR
  VAR_INPUT
        umax : REAL := 3.0000000000; (**)
  END_VAR
  VAR_INPUT
        T_filt_AI50 : REAL := 8.0000000000; (**)
  END_VAR
  VAR_INPUT
        invert : BOOL := TRUE; (**)
  END_VAR
  VAR_INPUT
        kp : REAL := 1.0000000000; (**)
  END_VAR
  VAR_INPUT
        ki : REAL := 1.0000000000; (**)
  END_VAR
  VAR_INPUT
        kd : REAL; (**)
  END_VAR
  VAR_INPUT
        N : REAL; (**)
  END_VAR
  VAR_INPUT
        Kt : REAL; (**)
  END_VAR
  VAR_INPUT
        deadband : REAL; (**)
  END_VAR
  VAR_INPUT
        uman : ARRAY[0..24] OF REAL; (*Reference Value*)
  END_VAR
  VAR_INPUT
        AI50ref : REAL; (*Reference Value*)
  END_VAR
  VAR_INPUT
        AI50offset : ARRAY[0..24] OF REAL; (*Reference Value*)
  END_VAR
  VAR_INPUT
        AI50offset_knck : ARRAY[0..24] OF REAL; (*Reference Value*)
  END_VAR
  VAR_INPUT
        K_knck : REAL := 1.0000000000; (*Gain for knocking IT offset*)
  END_VAR
  VAR_OUTPUT
        ITsat : ARRAY[0..24] OF REAL; (*IT saturation [°CA]*)
  END_VAR
  VAR_OUTPUT
        AI50err : ARRAY[0..24] OF REAL; (*AI50 error [°CA]*)
  END_VAR
  VAR_OUTPUT
        IToffset : ARRAY[0..24] OF REAL; (*IT offset [°CA]*)
  END_VAR
  VAR_OUTPUT
        DB_AI50_f : ARRAY[0..24] OF REAL; (*AI50 filtered*)
  END_VAR
  VAR_INPUT
        AI50_max : REAL := 30.0000000000; (*AI50 saturation max*)
  END_VAR
  VAR_INPUT
        AI50act : ARRAY[0..24] OF REAL; (*Reference Value*)
  END_VAR
  VAR_INPUT
        AI50_min : REAL; (*AI50 saturation min*)
  END_VAR
  VAR_OUTPUT
        dbg1 : ARRAY[0..5] OF REAL; (*u, utr, up, ui, ud, e*)
  END_VAR
  VAR_OUTPUT
        DB_Ts : LREAL; (**)
  END_VAR
	VAR
		bur_BlockIO_AI50toIT_mdl : BlockIO_AI50toIT_mdl;
	END_VAR
	VAR
		bur_D_Work_AI50toIT_mdl : D_Work_AI50toIT_mdl;
	END_VAR
	VAR
		bur_ExternalInputs_AI50toIT_mdl : ExternalInputs_AI50toIT_mdl;
	END_VAR
	VAR
		bur_ExternalOutputs_AI50toIT_md : ExternalOutputs_AI50toIT_mdl;
	END_VAR
END_FUNCTION_BLOCK
```

#### lAI50toIT.typ
```iecst
TYPE

END_TYPE
TYPE
BlockIO_AI50toIT_mdl : STRUCT
	Input16 : ARRAY[0..24] OF REAL;
	Input5 : REAL;
	Input8 : ARRAY[0..24] OF REAL;
	Input3 : ARRAY[0..24] OF REAL;
	Input4 : REAL;
	DiscreteTimeIntegrator : ARRAY[0..24] OF REAL;
	Product2 : ARRAY[0..24] OF REAL;
	Product1 : ARRAY[0..24] OF REAL;
	Integrator : ARRAY[0..24] OF REAL;
	Product4 : ARRAY[0..24] OF REAL;
	Switch2 : ARRAY[0..24] OF REAL;
	Modeswitch : ARRAY[0..24] OF REAL;
	Input1 : REAL;
	Input9 : ARRAY[0..24] OF REAL;
	Input2 : REAL;
END_STRUCT;
D_Work_AI50toIT_mdl : STRUCT
	DiscreteTimeIntegrator_DSTATE : ARRAY[0..24] OF REAL;
	Integrator_DSTATE : ARRAY[0..24] OF REAL;
	Filter_DSTATE : ARRAY[0..24] OF REAL;
	DiscreteTimeIntegrator_PrevRese : SINT;
END_STRUCT;
ExternalInputs_AI50toIT_mdl : STRUCT
	AI50act : ARRAY[0..24] OF REAL;
	AI50offset_knck : ARRAY[0..24] OF REAL;
END_STRUCT;
ExternalOutputs_AI50toIT_mdl : STRUCT
	IToffset : ARRAY[0..24] OF REAL;
	ITsat : ARRAY[0..24] OF REAL;
	AI50err : ARRAY[0..24] OF REAL;
END_STRUCT;
END_TYPE
```
